FUNCTION_BLOCK "GCS7_E_MZMN"	// FB 22
TITLE = MZAG/MZAH Flowbalancer
//  
//COPYRIGHT:    (C) 1997 BY  BUHLER AG, CH-9240 UZWIL  SWITZERLAND
//
//PRODUCT:      GCS7
//
//TITLE:        Element MZMN (Profibus) 
//
//-------------------------------------------------------------------------
//
//IDENT:        AUTHOR:             DEPT:                      DATE:
//
//FB22.5.2      A. Egli             BASE                       09-Apr-2008
//              Disable Alarm 18 Battery Low
//FB22.5.1      A.Egli              CT3                        01-Dec-2005
//              Parameter Upload Change DBD86-->DBD88
//FB22.5.0      A.Egli              CT3                        05-Jan-2005
//              Parameter Upload (uses DB10)
//FB22.4.2      A.Egli              CT3                        17-Nov-2003
//              - Alarm 90: Fault not RemoteControl
//              - Send RecipeNr=0 as long StStopped or StFault
//FB22.4.1      A.Egli              CT3                        03-Nov-2003
//              - in local mode Change to StStopped, when OutComFault
//FB22.4.0      A. Egli             CT3                        17-Jun-2002
//              MZMN Micro Dosing
//              LC Alarm 14 (DPFault) =Log Text number 12
//FB22.1A       A. Egli             CT3                        16-Apr-1998
//              1st Release in S7
//
//-------------------------------------------------------------------------
//
//PURPOSE:      MANUAL : see [MZGxxMAN]
//
//RESTRICTIONS: S7
//              ACCU2: Pointer to dynamic datas of the element
//              ACCU1: Pointer to parameter datas of the element
//
//=======================================================
//Log Message: 
//------------------------------------------------------
//0     = Fault Cannceled
//1..79 = AlarmLC : Alarmnumber see manual of MEAF
//90    = Fault Remote Control
//91    = StStopped
//92    = StDosing
//93    = StEmptied
//94    = Timeout starting
//95    = Wrong value
//96    = Communication fault
//97    = 
//98    = 
//99    = Collected alarm
//
//=======================================================
//StCode:  State               
//------------------------------------------------------
//32    StFault                 
// 1    StStopped                   Stopped
//41    Stopped.HWStop              StStopped + InHWStop 
//51    Stopped.DPFault             StStopped + DPFault
// 2    StStarting              
// 3    StStarted               
// 7    StStopping              
//
AUTHOR : EA
FAMILY : GCS7LL
NAME : MZMN
VERSION : 5.1
VAR
  StCode : INT ;	//Element state code
  InEnable : BOOL ;	//Enable to run the element (manual and automatic mode)
  spare21 : BOOL ;
  spare22 : BOOL ;
  spare23 : BOOL ;
  CmdNewValue : BOOL ;	//Send new target values
  spare25 : BOOL ;
  spare26 : BOOL ;
  spare27 : BOOL ;
  CmdOff : BOOL ;	//Pulse to stop the element (manual mode)
  CmdOn : BOOL ;	//Pulse to start the element (manual mode)
  CmdNext : BOOL ;	//Pulse to start the element in automatic mode
  CmdFaultReset : BOOL ;	//Command to reset fault
  InLocal : BOOL ;	//1= Local mode (no fault by start with service switch)
  InManual : BOOL ;	//1= Manual / 0= Automatic
  InReport : BOOL ;	//Report of all state transitions
  spare0307 : BOOL ;
  InHWStop : BOOL ;	//HW stop is detected, no fault
  InDPFault : BOOL ;	//DP-Fault is detected, no fault
  InSimulation : BOOL ;	//Simulation with DPSim
  OutComFault : BOOL ;	//Communication fault
  spare44 : BOOL ;
  spare45 : BOOL ;
  spare46 : BOOL ;
  spare47 : BOOL ;
  StStopped : BOOL ;	//Element is stopped
  StStarting : BOOL ;	//Element is starting
  StStarted : BOOL ;	//Element is dosing
  StStopping : BOOL ;	//Element is stopping
  StFault : BOOL ;	//Element has a communication or device fault
  spare55 : BOOL ;
  spare56 : BOOL ;
  spare57 : BOOL ;
  InFlowrate : DINT ;	//Flowrate target value [0.1%]
  InRecipeNr : INT ;	//Is send to LC
  OutFlowrate : DINT ;	//Is read from LC [10g/h]
  OutRecipeNr : INT ;	//Is read from MEAF
  OutLCStep : INT ;	//Is read from MEAF
  OutAlarmNr : INT ;	//Is read from MEAF
  OutAlarmNrLog : INT ;	//Last textnumber send to log
  RecipeMZMN : STRUCT
   InRecipeNr : INT ;	//Recipe to read or write
   CmdSend : BOOL ;	//1= Send Dataset 136
   CmdRead : BOOL ;	//1= Read Dataset 136
   OutSendDone : BOOL ;	//Send is done
   OutReadDone : BOOL ;	//Read is done
   OutWrongValue : BOOL ;	//MEAF has recipe rejected
   Desity : INT ;	//de: Spezifisches Gewicht REC.DENS
   CorrectionFactor : INT ;	//de: Korrekturfactor REC.FACT
   NominalRate : INT ;	//de: Sollleistung REC.FLOS
   MixerFrequency : INT ;	//de: Frequenz Wirbler REC.MIX
   TypeRate : INT ;	//de: Volumetrische Typenleistung REC:FTYP
   AgitatorCutoutMode : INT ;	//de: Aussetzbetrieb Rührwerk REC.IOFF
   spare16 : INT ;
   spare18 : INT ;
  END_STRUCT ;
  Par : STRUCT
   ParObjectNo : INT ;	//Is used for communication with PC, e.g. for message
   ParMsgType : INT ;	//Is used for message (translation of state)
   ParHornCode : INT ;	//Is used by horn module
   ParLogOff : BOOL ;	//Report is off
   ParManual : BOOL ;	//Manual mode wihout interlocking
   ParFilter : STRUCT 	//Filter to alarm 1=Ignore alarm
    SumFault : BOOL ;	//de: Sammelalarm
    A05_24VToLow : BOOL ;
    A07ADRange : BOOL ;
    A08ADCalibration : BOOL ;
    A09ADFunction : BOOL ;
    A10ADSupply : BOOL ;
    A11AnalogInput : BOOL ;
    A12SerialInterface : BOOL ;
    A13RemoteControl : BOOL ;
    A16Printer : BOOL ;
    A25FrequenceConverter : BOOL ;
    A54Relais : BOOL ;
   END_STRUCT ;
   ParIOByteNr : INT ;	//PROFIBUS: Address of first input and output byte
   ParMonTime : INT ;	//Monitoring time starting and stopping
   OutMonTime : INT ;	//Monitoring time starting and stopping
   HelpFlags : STRUCT
    OutAlarmTimeOut : BOOL ;
    CmdNewValue : BOOL ;
    CmdFaultReset : BOOL ;
    OutFaultResetDone : BOOL ;
    OutTestNewAlarm : BOOL ;	//Aux. signal to retry fault message
    spare0007 : BOOL ;
    OutRelevantFault : BOOL ;
    OutNoAlarm : BOOL ;	//Alarmnumber 0 is read form LC
    OutFlagFaultResetDone : BOOL ;
    OutComFaultRead : BOOL ;
    OutComFaultSend : BOOL ;
   END_STRUCT ;
   Command : STRUCT
    Start : BOOL ;	//de: Start
    spare01 : BOOL ;
    spare02 : BOOL ;
    spare03 : BOOL ;
    spare04 : BOOL ;
    spare05 : BOOL ;
    spare06 : BOOL ;
    AcceptNewDataReady : BOOL ;	//de: Quittierung neue Werte Bereit
    spare10 : BOOL ;
    Recipe1 : BOOL ;	//MZMN: Command to select recipe 1
    Recipe2 : BOOL ;	//MZMN: Command to select recipe 2
    Recipe3 : BOOL ;	//MZMN: Command to select recipe 3
    Recipe4 : BOOL ;	//MZMN: Command to select recipe 4
    Recipe5 : BOOL ;	//MZMN: Command to select recipe 5
    Recipe6 : BOOL ;	//MZMN: Command to select recipe 6
    spare20 : BYTE ;
    CommandReady : BOOL ;	//de: Steuersignale gültig
    spare31 : BOOL ;
    spare32 : BOOL ;
    spare33 : BOOL ;
    spare34 : BOOL ;
    ResetAlarm : BOOL ;	//de: Alarm löschen
    NewSendData : BOOL ;	//de: Aenderung Sendedaten
    AcceptNewRcvData : BOOL ;	//de: Quittierung Aenderung Empfangsdatensatz
   END_STRUCT ;
   Status : STRUCT
    Operation : BOOL ;	//de: Betrieb
    spare01 : BOOL ;
    spare02 : BOOL ;
    spare03 : BOOL ;
    spare04 : BOOL ;
    spare05 : BOOL ;
    spare06 : BOOL ;
    NewDataReady : BOOL ;	//de: Neue Werte Bereit
    spare10 : BOOL ;
    Recipe1 : BOOL ;	//MZMN2 , Recipe 2 is active
    Recipe2 : BOOL ;	//MZMN3 , Recipe 3 is active
    Recipe3 : BOOL ;	//MZMN3 , Recipe 3 is active
    Recipe4 : BOOL ;	//MZMN4 , Recipe 4 is active
    Recipe5 : BOOL ;	//MZMN5 , Recipe 5 is active
    Recipe6 : BOOL ;	//MZMN6 , Recipe 6 is active
    spare20 : BYTE ;
    spare30 : BOOL ;
    spare31 : BOOL ;
    spare32 : BOOL ;
    RemoteControl : BOOL ;	//de: Sollwertvorgabe Remote
    WrongValue : BOOL ;	//de: Falscher Sollwert
    SumFault : BOOL ;	//de: Sammelalarm
    AcceptNewSendData : BOOL ;	//de: Quittierung Aenderung Sendedaten
    NewRcvData : BOOL ;	//de: Aenderung Empfangsdaten
   END_STRUCT ;
  END_STRUCT ;
END_VAR
VAR_TEMP
  tmpLOGvalue : WORD ;	//LOG value
  tmpCommand : INT ;
  tmpFault : BOOL ;
  tmpOff : BOOL ;
  tmpOn : BOOL ;
  tmpLocal : BOOL ;
  tmpLocalFault : BOOL ;
  tmpReport : BOOL ;
  tmpFlag : BOOL ;
  tmpLenDyn : DINT ;
  tmpAddrOutComFlags : DWORD ;	//Pointer to OutComFlags
  tmpWt : DINT ;
  tmpFilter : ARRAY  [0 .. 100 ] OF BOOL ;
  tmpAddrOffset : DINT ;
  tmpAddr : WORD ;
  tmpReturn : INT ;
  DPData : STRUCT
   StatusCommand : DWORD ;
   NrSndDataSet : BYTE ;	//de: Nummer Sendedatensatz
   IdxSndDataSet : BYTE ;	//de: Index Sendedatensatz
   NrRcvDataSet : BYTE ;	//de: Nummer Empfangsdatensatz
   IdxRcvDataSet : BYTE ;	//de: Index Empfangsdatensatz
   Data : ARRAY  [1 .. 4 ] OF DINT ;
  END_STRUCT ;
  Set001 : STRUCT
   FlowrateAc : DINT ;	//de: Istleistung kg/h
   spare4 : DINT ;	//de: Isttotalgewicht kg
   spare8 : DINT ;	//de: nochtlöschbarese Totalgewicht
   spare12 : BYTE ;
   RecipeNr : BYTE ;
   Step : BYTE ;
   AlarmNr : BYTE ;
  END_STRUCT ;
  tmpHornOn : BOOL ;
END_VAR
BEGIN
NETWORK
TITLE =  Start Global
      L     70;
      T     #tmpLenDyn;	//--> Len dynamic data in byte
      SET;
      R     #tmpHornOn;
NETWORK
TITLE = Filter
      LAR1  P##tmpFilter;
      L     0;
      T     D [AR1,P#0.0];	//tmpFilter[00..31]
      T     D [AR1,P#0.0];	//tmpFilter[32..63]
      T     D [AR1,P#0.0];	//tmpFilter[64..95]
      SET;	//[4.1]
      =     #tmpFilter[0];
      A     #Par.ParFilter.A05_24VToLow;
      =     #tmpFilter[5];
      A     #Par.ParFilter.A07ADRange;
      =     #tmpFilter[7];
      A     #Par.ParFilter.A08ADCalibration;
      =     #tmpFilter[8];
      A     #Par.ParFilter.A09ADFunction;
      =     #tmpFilter[9];
      A     #Par.ParFilter.A10ADSupply;
      =     #tmpFilter[10];
      A     #Par.ParFilter.A11AnalogInput;
      =     #tmpFilter[11];
      A     #Par.ParFilter.A12SerialInterface;
      =     #tmpFilter[12];
      =     #tmpFilter[14];	//[4.0]
      A     #Par.ParFilter.A13RemoteControl;
      =     #tmpFilter[13];
      A     #Par.ParFilter.A16Printer;
      =     #tmpFilter[16];
      SET;
      =     #tmpFilter[18];	//[5.2] Battery Low
      A     #Par.ParFilter.A25FrequenceConverter;
      =     #tmpFilter[25];
      A     #Par.ParFilter.A54Relais;
      =     #tmpFilter[54];
NETWORK
TITLE = PC Control
//=== Test Object number =====================
      L     "SYS_DirectCtrlDB".PC.ObjectNo;	//PCControl.ObjectNo
      L     #Par.ParObjectNo;	//Input ObjectNo
      <>I;
      JC    Ctrl;
//=== Test OType      ========================
      L     1022;	//Input object type
      L     "SYS_DirectCtrlDB".PC.ObjectType;	//PCControl.ObjectType
      <>I;
      JC    Ctrl;
//=== Test Handshake =========================
      A     "SYS_DirectCtrlDB".PC.Hsk.FExamine;	//Handshake.FExamine
      JC    pExa;
      A     "SYS_DirectCtrlDB".PC.Hsk.FDefineCmd;	//Handshake.FDefineCmd
      JC    pCmd;
      A     "SYS_DirectCtrlDB".PC.Hsk.FDefinePara;	//Handshake.FDefinePara
      JC    pPar;
pIni: L     2;	//FcInit
      UC    "SYS_DirectCtrl";
      JU    Ctrl;
// Write parameter 
pPar: LAR1  P#DBX 58.0;
      L     P##Par;
      L     DW#16#FFFFF;
      AD;
      +AR1;
      L     DBD [AR1,P#12.0];
      T     #Par.ParMonTime;
//Write new commands from PC to Interface of group 
pCmd: A     "SYS_DirectCtrlDB".PC.Cmd1[4];	//Cmd1[4]  =CmdNewValue
      S     #CmdNewValue;
      A     "SYS_DirectCtrlDB".PC.Cmd1[8];	//Cmd1[8]  =CmdOff
      S     #CmdOff;
      A     "SYS_DirectCtrlDB".PC.Cmd1[9];	//Cmd1[9]  =CmdOn
      S     #CmdOn;
      A     "SYS_DirectCtrlDB".PC.Cmd1[10];	//Cmd1[10] =CmdNext
      S     #CmdNext;
      A     "SYS_DirectCtrlDB".PC.Cmd1[11];	//Cmd1[11] =CmdFaultReset
      S     #CmdFaultReset;
      A     "SYS_DirectCtrlDB".PC.Cmd1[13];	//Cmd1[13] =CmdManualOn
      S     #InManual;
      A     "SYS_DirectCtrlDB".PC.Cmd2[13];	//Cmd2[13] =CmdManualOff
      R     #InManual;
      A     "SYS_DirectCtrlDB".PC.Cmd1[14];	//Cmd1[14] =CmdReportOn
      S     #InReport;
      A     "SYS_DirectCtrlDB".PC.Cmd2[14];	//Cmd2[14] =CmdReportOff
      R     #InReport;
//Define Value
      AN    "SYS_DirectCtrlDB".PC.Hsk.FDefineValue;	// PC.Hsk.FDefineValue
      ON    #InManual;
      JC    pIni;
      LAR1  P#DBX 58.0;
      L     DBD [AR1,P#6.0];
      T     #InFlowrate;
      L     DBW [AR1,P#10.0];
      T     #InRecipeNr;
      JU    pIni;
pExa: TAR2;	//Address dynamic datas
      T     "SYS_DirectCtrlDB".GC.InDynAddr;	//-->PCControl.GC.InDynAddr
      L     #tmpLenDyn;	//Length dynamic datas
      T     "SYS_DirectCtrlDB".GC.InDynLen;	//-->PCControl.GC.InDynLen
      L     0;
      T     "SYS_DirectCtrlDB".GC.InParaAddr;	//-->PCControl.GC.InParaAddr
      T     "SYS_DirectCtrlDB".GC.InParaLen;	//-->PCControl.GC.InParaLen
      L     1;	//Code FcExamine
      UC    "SYS_DirectCtrl";
      L     10;	//Revision
      T     "SYS_DirectCtrlDB".GC.Revision;
Ctrl: NOP   0;
NETWORK
TITLE = (Profibus) Read data and store Data 
      L     #Par.ParIOByteNr;
      T     #tmpAddr;
      A     #InSimulation;
      JC    rSim;
      CALL  "SIEMENS_DPRD_DAT" (
           LADDR                    := #tmpAddr,
           RET_VAL                  := #tmpReturn,
           RECORD                   := #DPData);
      L     #tmpReturn;
      L     0;
      <>I;
      =     #Par.HelpFlags.OutComFaultRead;
      JC    rcv0;
      JU    rDP;
//read from Simulation
rSim: R     #Par.HelpFlags.OutComFaultRead;
      A     "GCS7_Gr_SimDPtoImage";
      L     P#I 0.0;
      JC    rDB1;
      OPN   "TEST_IOSimuliInput";
      L     P#DBX 0.0;
rDB1: L     #Par.ParIOByteNr;
      SLD   3;
      +D;
      LAR1;
      L     D [AR1,P#0.0];
      T     #DPData.StatusCommand;
      L     B [AR1,P#4.0];
      T     #DPData.NrSndDataSet;
      L     B [AR1,P#5.0];
      T     #DPData.IdxSndDataSet;
      L     B [AR1,P#6.0];
      T     #DPData.NrRcvDataSet;
      L     B [AR1,P#7.0];
      T     #DPData.IdxRcvDataSet;
      L     D [AR1,P#8.0];
      T     #DPData.Data[1];
      L     D [AR1,P#12.0];
      T     #DPData.Data[2];
      L     D [AR1,P#16.0];
      T     #DPData.Data[3];
      L     D [AR1,P#20.0];
      T     #DPData.Data[4];
//==Copy Status===============
rDP:  L     #DPData.NrRcvDataSet;
      L     0;
      ==I;
      JC    R001;
      CALL  "SIEMENS_BLKMOV" (
           SRCBLK                   := #DPData.StatusCommand,
           RET_VAL                  := #tmpReturn,
           DSTBLK                   := #Par.Status);
      AN    #Par.Status.NewRcvData;
      A     #InSimulation;
      JC    rcv0;
//===============================
//Answer Dataset 001
      L     #DPData.NrRcvDataSet;
      L     1;
      <>I;
      JC    r11;	//[5.0]
      CALL  "SIEMENS_BLKMOV" (
           SRCBLK                   := #DPData.Data,
           RET_VAL                  := #tmpReturn,
           DSTBLK                   := #Set001);
      L     #Set001.FlowrateAc;
      T     #OutFlowrate;
      L     #Set001.RecipeNr;
      T     #OutRecipeNr;
      L     #Set001.Step;
      T     #OutLCStep;
//Reset old alarm flags with CmdFaultReset
      A     #Par.HelpFlags.OutFlagFaultResetDone;
      A     "SYS_Pulse1000ms";
      R     #Par.HelpFlags.OutFlagFaultResetDone;
      R     #Par.HelpFlags.OutFaultResetDone;
      S     #Par.HelpFlags.OutTestNewAlarm;
      L     0;
      L     #Set001.AlarmNr;
      ==I;
      =     #Par.HelpFlags.OutNoAlarm;
      <>I;
      O     #Par.ParFilter.SumFault;
      =     #tmpFilter[0];
//  keep old alalrm number
      A     #Par.HelpFlags.OutNoAlarm;
      A     #Par.HelpFlags.OutRelevantFault;
      AN    #Par.HelpFlags.OutTestNewAlarm;
      AN    #InLocal;
      AN    #InManual;
      JC    rA1;
      T     #OutAlarmNr;
rA1:  JU    R11;	//[5.0]
//===============================
//[5.0]--> LC Parameter 
//Reading dataset 11
R11:  L     "SYS_DirectCtrlLCDB".PC.ObjectNo;
      L     #Par.ParObjectNo;
      <>I;
      JC    R127;
      AN    "SYS_DirectCtrlLCDB".PC.Hsk.FExamineFirst;
      AN    "SYS_DirectCtrlLCDB".PC.Hsk.FExamineNext;
      JC    R127;
// -- Start Reading with Dataset 11
      L     11;
      T     #DPData.NrRcvDataSet;
      L     253;	//First
      A     "SYS_DirectCtrlLCDB".PC.Hsk.FExamineFirst;
      JC    rLC9;
      L     254;	//Next
rLC9: T     #DPData.IdxRcvDataSet;
      JU    rcv0;
//---Answer  dataset 11 ---
//---Answer  dataset 12 ---
r11:  L     #DPData.NrRcvDataSet;
      L     11;
      <>I;
      JC    rLCB;
// Answer Dataset 11
      L     '  ';
      T     "SYS_DirectCtrlLCDB".PC.Value[1];
      L     #DPData.Data[1];
      T     DB10.DBD 60;
      L     #DPData.Data[2];
      T     DB10.DBD 64;
      L     #DPData.Data[3];
      T     DB10.DBD 68;
      L     #DPData.Data[4];
      T     DB10.DBD 72;
      L     #DPData.IdxRcvDataSet;
      L     255;
      ==I;
      JC    rLCE;
      S     "SYS_DirectCtrlLCDB".GC.Set11Done;
      L     12;
      T     #DPData.NrRcvDataSet;
      L     0;
      T     #DPData.IdxRcvDataSet;
      JU    rcv0;	//--> Read dataset 12
// Answer Dataset 12
rLCB: L     #DPData.NrRcvDataSet;
      L     12;
      <>I;
      JC    r127;
      L     #DPData.Data[1];
      T     DB10.DBD 76;
      L     #DPData.Data[2];
      T     DB10.DBD 80;
      L     #DPData.Data[3];
      T     DB10.DBD 84;
      L     #DPData.Data[4];
      T     DB10.DBD 88;
      AN    "SYS_DirectCtrlLCDB".GC.Set11Done;
      JC    R127;
rLCE: L     12;
      CALL  "SYS_DirectCtrl";
      JU    R127;
//<--[5.0]
//===============================
//Answer  dataset 127
r127: L     #DPData.NrRcvDataSet;
      L     127;
      <>I;
      JC    r128;
      JU    R128;
//===============================
//Answer  dataset 128
r128: JU    r136;
//===============================
//Answer  dataset 136
r136: L     #DPData.NrRcvDataSet;
      L     136;
      <>I;
      JC    R001;	// =no valide answer read dataset 001
      L     #RecipeMZMN.InRecipeNr;
      L     #DPData.IdxRcvDataSet;
      ==I;
      JCN   R001;
      R     #RecipeMZMN.CmdRead;
      S     #RecipeMZMN.OutReadDone;
      L     #DPData.Data[1];
      T     #RecipeMZMN.CorrectionFactor;
      SRD   16;
      T     #RecipeMZMN.Desity;
      L     #DPData.Data[2];
      T     #RecipeMZMN.NominalRate;
      L     #DPData.Data[3];
      T     #RecipeMZMN.TypeRate;
      SRD   16;
      T     #RecipeMZMN.MixerFrequency;
      L     #DPData.Data[4];
      L     W#16#FFFF;
      AW;
      SRD   8;
      T     #RecipeMZMN.AgitatorCutoutMode;
      JU    R001;
//===============================
//Read Dataset 001
R001: L     1;
      T     #DPData.NrRcvDataSet;
      L     0;
      T     #DPData.IdxRcvDataSet;
      A     #Par.HelpFlags.OutFaultResetDone;
      AN    "SYS_Pulse1000ms";
      S     #Par.HelpFlags.OutFlagFaultResetDone;
      JU    rcv0;
//===============================
//Read Dataset 127
R127: L     127;
      T     #DPData.NrRcvDataSet;
      L     0;
      T     #DPData.IdxRcvDataSet;
      JU    rcv0;
//===============================
//Read Dataset 128
R128: JU    R136;
//===============================
//Read Dataset 136
R136: AN    #RecipeMZMN.CmdRead;
      JC    R001;
      L     136;
      T     #DPData.NrRcvDataSet;
      L     #RecipeMZMN.InRecipeNr;
      T     #DPData.IdxRcvDataSet;
      JU    rcv0;
//===============================
rcv0: NOP   0;
      NOP   0;
NETWORK
TITLE = (Profibus) Status to ASW
      A     #Par.HelpFlags.OutComFaultRead;
      O     #Par.HelpFlags.OutComFaultSend;
      =     #OutComFault;
//=======================================
//Init in local mode  
//=======================================
      AN    #InLocal;
      AN    #InManual;
      ON    #OutComFault;
      JC    alJL;
      L     0;
      T     #OutFlowrate;
alJL: NOP   0;
      NOP   0;
NETWORK
TITLE =  All State Init
//===Clear tmp Variable
//===Global Group Orders===
      A     "GCS7_Gr_OutManualOn";	//Global.OutManualOn
      S     #InManual;
      A     "GCS7_Gr_OutManualOff";	//Global.OutManualOff
      R     #InManual;
      A     #InManual;
      S     "GCS7_Gr_InManual";	//Global.InManualMode
//---Report is on---
      O     "GCS7_Gr_OutReportAll";	//---Global OutReportAll
      O     #InReport;
      =     #tmpReport;
//---FaultReset is on---
      A     "GCS7_Gr_OutFaultReset";	//Gr.OutFaultReset
      S     #CmdFaultReset;
//---Local---
      A     #InLocal;
      AN    #InManual;
      =     #tmpLocalFault;
      A     #tmpLocalFault;
      O     #InHWStop;
      O     #InDPFault;
      =     #tmpLocal;
//---Off---
      AN    #InManual;
      ON    #Par.ParManual;
      AN    #InEnable;
      O     #tmpLocal;
      O     #CmdOff;
      =     #tmpOff;
//---On---
      A     #CmdNext;
      AN    #InManual;
      O     #CmdOn;
      AN    #tmpOff;
      =     #tmpOn;
//--- Send Recipe
      A     #RecipeMZMN.CmdSend;
      R     #RecipeMZMN.OutSendDone;
//--- Read Recipe
      A     #RecipeMZMN.CmdRead;
      R     #RecipeMZMN.OutReadDone;
//--- tmpFault   
// Time out
      AN    #StStarting;
      AN    #StStopping;
      AN    #StFault;
      R     #Par.HelpFlags.OutAlarmTimeOut;
      JC    inJ1;
      A     #Par.HelpFlags.OutAlarmTimeOut;
      O     #StFault;
      JC    inJ1;
      L     0;
      L     #Par.OutMonTime;
      >I;
      =     #Par.HelpFlags.OutAlarmTimeOut;
      AN    "GCS7_Gr_OutTick200ms";	// Global Tick 200ms
      JC    inJ1;
      +     -2;	// Decrement all 200ms
      T     #Par.OutMonTime;
inJ1: NOP   0;
//=======================================
//Fault   
//=======================================
      LAR1  P##tmpFilter;
      L     #OutAlarmNr;
      +AR1;	//Pointer to #tmpFilter[OutAlarmNumber]
      L     #OutAlarmNr;
      L     0;
      <>I;
      AN    L [AR1,P#0.0];	//#tmpFilter[OutAlarmNumber]
      =     #Par.HelpFlags.OutRelevantFault;
      A     #Par.HelpFlags.OutRelevantFault;
      O     #OutComFault;
      O     #Par.HelpFlags.OutAlarmTimeOut;
      O     #Par.Status.WrongValue;
      ON    #Par.Status.RemoteControl;	//[4.2]
      AN    #tmpLocal;
      =     #tmpFault;
      NOP   0;
NETWORK
TITLE = (Profibus) Prepare Command for MEAF
//==============================
      A     #Par.Status.AcceptNewSendData;
      A     #Par.Command.ResetAlarm;
      R     #Par.Command.ResetAlarm;
      S     #Par.HelpFlags.OutFaultResetDone;
      A     #CmdFaultReset;
      AN    #Par.Status.AcceptNewSendData;
      R     #CmdFaultReset;
      S     #Par.Command.ResetAlarm;
      R     #Par.HelpFlags.OutAlarmTimeOut;
//================================
      A     #tmpOn;
      AN    #Par.HelpFlags.CmdNewValue;
      S     #Par.Command.Start;
      A     #StFault;
      A     #Par.HelpFlags.OutNoAlarm;
      O     #tmpOff;
      R     #Par.Command.Start;
//==============================
      A     #Par.Status.NewDataReady;
      =     #Par.Command.AcceptNewDataReady;
//==============================
      SET;
      =     #Par.Command.CommandReady;
//==============================
      A     #Par.Status.NewRcvData;
      =     #Par.Command.AcceptNewRcvData;
//==============================
      AN    #Par.Status.AcceptNewSendData;
      =     #Par.Command.NewSendData;
//==============================
//Command MZMN 
      L     #InRecipeNr;
      L     1;
      ==I;
      =     #Par.Command.Recipe1;
      L     #InRecipeNr;
      L     2;
      ==I;
      =     #Par.Command.Recipe2;
      L     #InRecipeNr;
      L     3;
      ==I;
      =     #Par.Command.Recipe3;
      L     #InRecipeNr;
      L     4;
      ==I;
      =     #Par.Command.Recipe4;
      L     #InRecipeNr;
      L     5;
      ==I;
      =     #Par.Command.Recipe5;
      L     #InRecipeNr;
      L     6;
      ==I;
      =     #Par.Command.Recipe6;
      NOP   0;
NETWORK
TITLE = (Profibus) Send Data
//======================================================
//Test Send Dataset 000 done
      L     #DPData.NrSndDataSet;
      L     0;
      <>I;
      JC    s128;
      JU    S128;	//-->send 128
//------------------------------------------------
//Test Send Dataset 128 done
s128: L     #DPData.NrSndDataSet;
      L     128;
      <>I;
      JC    s136;
      AN    #Par.Status.WrongValue;
      A     #Par.HelpFlags.CmdNewValue;
      A     #CmdNewValue;
      R     #Par.HelpFlags.CmdNewValue;
      R     #CmdNewValue;
      JU    S136;	//-->Send 136
//------------------------------------------------
//Test Send Dataset 136 done
s136: L     #DPData.NrSndDataSet;
      L     136;
      <>I;
      JC    S000;
      L     #DPData.IdxSndDataSet;
      L     #RecipeMZMN.InRecipeNr;
      ==I;
      JCN   S128;	//-->Send 128
      A     #Par.Status.WrongValue;
      S     #RecipeMZMN.OutWrongValue;
      AN    #Par.Status.WrongValue;
      R     #RecipeMZMN.CmdSend;
      S     #RecipeMZMN.OutSendDone;
      R     #RecipeMZMN.OutWrongValue;
      JU    S128;	//-->Send 128
//==================================================
//Send Dataset 128
S128: A     #CmdNewValue;
      =     #Par.HelpFlags.CmdNewValue;
      L     128;
      T     #DPData.NrSndDataSet;
      L     0;
      T     #DPData.IdxSndDataSet;
      L     #InFlowrate;
      SLD   16;
      T     #DPData.Data[1];
      L     0;
      T     #DPData.Data[2];
      L     0;
      T     #DPData.Data[3];
      A     #StStopped;	//[4.2]
      O     #StFault;	//[4.2]
      L     0;	//[4.2]
      JC    snJ8;	//[4.2]
      L     #InRecipeNr;
      SLD   16;
snJ8: T     #DPData.Data[4];	//-->Byte 21
      JU    send;
//======================================================
//Send Dataset 136
S136: AN    #RecipeMZMN.CmdSend;
      JC    S000;
      L     136;
      T     #DPData.NrSndDataSet;
      L     #RecipeMZMN.InRecipeNr;
      T     #DPData.IdxSndDataSet;
      L     #RecipeMZMN.Desity;
      SLD   16;
      L     #RecipeMZMN.CorrectionFactor;
      OD;
      T     #DPData.Data[1];
      L     #RecipeMZMN.NominalRate;
      T     #DPData.Data[2];
      L     #RecipeMZMN.MixerFrequency;
      SLD   16;
      L     #RecipeMZMN.TypeRate;
      OD;
      T     #DPData.Data[3];
      L     #RecipeMZMN.AgitatorCutoutMode;
      SLD   8;
      T     #DPData.Data[4];
      JU    send;
//======================================================
//Send Dataset 0
S000: L     0;
      T     #DPData.NrSndDataSet;
      L     0;
      T     #DPData.IdxSndDataSet;
send: CALL  "SIEMENS_BLKMOV" (
           SRCBLK                   := #Par.Command,
           RET_VAL                  := #tmpReturn,
           DSTBLK                   := #DPData.StatusCommand);
      A     #InSimulation;
      JC    sSim;
      CALL  "SIEMENS_DPWR_DAT" (
           LADDR                    := #tmpAddr,
           RECORD                   := #DPData,
           RET_VAL                  := #tmpReturn);
      L     #tmpReturn;
      L     0;
      <>I;
      =     #Par.HelpFlags.OutComFaultSend;
      JU    DP_C;
//write to Simulation
sSim: R     #Par.HelpFlags.OutComFaultSend;
      A     "GCS7_Gr_SimDPtoImage";
      L     P#Q 0.0;
      JC    rDB2;
      OPN   "TEST_IOSimuliOutput";
      L     P#DBX 0.0;
rDB2: L     #Par.ParIOByteNr;
      SLD   3;
      +D;
      LAR1;
      L     #DPData.StatusCommand;
      T     D [AR1,P#0.0];
      L     #DPData.NrSndDataSet;
      T     B [AR1,P#4.0];
      L     #DPData.IdxSndDataSet;
      T     B [AR1,P#5.0];
      L     #DPData.NrRcvDataSet;
      T     B [AR1,P#6.0];
      L     #DPData.IdxRcvDataSet;
      T     B [AR1,P#7.0];
      L     #DPData.Data[1];
      T     D [AR1,P#8.0];
      L     #DPData.Data[2];
      T     D [AR1,P#12.0];
      L     #DPData.Data[3];
      T     D [AR1,P#16.0];
      L     #DPData.Data[4];
      T     D [AR1,P#20.0];
DP_C: NOP   0;
NETWORK
TITLE = States
//===State machine===
      A     #StStopped;
      JC    S0;
      A     #StStarting;
      JC    S1;
      A     #StStarted;
      JC    S2;
      A     #StStopping;
      JC    S3;
      A     #StFault;
      JC    S4;
      S     #StStopped;	//Init
      JU    S0;
NETWORK
TITLE =  StStopped
xxS0: S     #StStopped;
      R     #StStarted;
      JU    LOGX;
S0:   A     #tmpFault;
      S     #tmpHornOn;
      R     #StStopped;
      JC    xxS4;	////--> Transition to StFault
      A     #tmpOn;
      O     #Par.Status.Operation;
      AN    #OutComFault;	//[4.1]
      R     #StStopped;
      JC    xxS1;	//--> Transition to StStarting
      JU    OUT;
NETWORK
TITLE =  StStarting
xxS1: S     #StStarting;
      R     #Par.HelpFlags.OutAlarmTimeOut;
      L     #Par.ParMonTime;
      T     #Par.OutMonTime;
      JU    OUT;
S1:   A     #tmpFault;	//Condition for StFault
      R     #StStarting;
      JC    xxS4;	//--> Transition to StFault
      A     #tmpOff;
      R     #StStarting;
      JC    xxS3;	//--> Transition to StStopping
      A     #Par.Status.Operation;
      R     #StStarting;
      JC    xxS2;	//--> Transition to StStarted
      JU    OUT;
NETWORK
TITLE =  StStarted
xxS2: S     #StStarted;
      R     #StStopped;
      JU    LOGX;
S2:   A     #tmpFault;	//Condition for StFault/StFalse
      S     #tmpHornOn;
      R     #StStarted;
      JC    xxS4;	//--> Transition to StFault
      A     #tmpOff;
      ON    #Par.Status.Operation;
      O     #OutComFault;	//[4.1]
      R     #StStarted;
      JC    xxS3;	//--> Transition to StStopping
      JU    OUT;
NETWORK
TITLE =  StStopping
xxS3: S     #StStopping;
      R     #Par.HelpFlags.OutAlarmTimeOut;
      L     #Par.ParMonTime;
      T     #Par.OutMonTime;
      A     #StFault;
      R     #StFault;
      JC    LOGC;	//-->Message Operator ('fault cancelled' )
//-----------------------------------
//--> Transition to StFault
S3:   A     #tmpFault;
      AN    #tmpLocal;
      S     #tmpHornOn;
      R     #StStopping;
      JC    xxS4;	//-->Transition to StFault
//-----------------------------------
//--> Transition to StStarting
      A     #tmpOn;
      R     #StStopping;
      JC    xxS1;	//-->Transition to StStarting 
//-----------------------------------
//--> Transition to StStopped
      AN    #tmpFault;	//Transition to StFaulte
      AN    #Par.Status.Operation;
      O     #OutComFault;	//[4.1]
      R     #StStopping;
      JC    xxS0;	//-->Transition to StStopped 
      JU    OUT;
NETWORK
TITLE =  FAULT
// State Fault
S4:   AN    #tmpFault;	//---Condition for StStopping
      A     #Par.HelpFlags.OutTestNewAlarm;
      O     #tmpLocalFault;
      JC    xxS3;	// Transition to StStopping
      A     #Par.HelpFlags.OutTestNewAlarm;
      JC    xxS4;
      JU    OUT;
NETWORK
TITLE = LOG
xxS4: S     #tmpHornOn;
      S     #StFault;
      R     #Par.HelpFlags.OutFaultResetDone;
      R     #Par.HelpFlags.OutTestNewAlarm;
      L     #Par.ParMonTime;
      T     #Par.OutMonTime;
//Alarm Communication
      L     B#(1, 96);
      A     #OutComFault;
      JC    LOG;
//Tiemout
      A     #Par.HelpFlags.OutAlarmTimeOut;
      L     B#(1, 94);	// Message ('fault timeout')
      JC    LOG;
//Alarm-Nr 1..80
      L     0;
      L     #OutAlarmNr;
      ==I;
      JC    LOG2;
      L     B#(1, 0);
      OW;
      JU    LOG;	//Alarms 1..80
//Fault Wrong Value
LOG2: L     B#(1, 90);	// Message ('fault DP Mode')   //[4.2]
      AN    #Par.Status.RemoteControl;	//[4.2]
      JC    LOG;	//[4.2]
//Fault Wrong Value
      A     #Par.Status.WrongValue;
      L     B#(1, 95);	// Message ('fault wrong value')
      JC    LOG;
//Collected Alarm
      L     B#(1, 99);	// Message ('fault collected alarm')
      JU    LOG;
//===============================================
//State Transition
LOGX: AN    #tmpReport;
      JC    OUT;
      A     #StStopped;
      L     B#(4, 91);	//Message ('Stopped')
      JC    LOG;
      A     #StStarted;
      L     B#(4, 92);	//Message ('Dosing')
      JC    LOG;
      JU    OUT;
LOGC: L     B#(4, 0);	//Message ('fault cancelled')
LOG:  A     #Par.ParLogOff;	//---Set LOG Message
      JC    SAVE;
      T     #tmpLOGvalue;
      L     W#16#FF;
      AW;
      T     #OutAlarmNrLog;
      CALL  "GCS7_LogConvert" (
           ObjectNo                 := #Par.ParObjectNo,
           MsgType                  := #Par.ParMsgType,
           ClassMsgTxt              := #tmpLOGvalue,
           OType                    := 1026);	//LOG Message Converter / Entry / Contains Class and TextNo
SAVE: NOP   0;
OUT:  NOP   0;
NETWORK
TITLE = Global End
      SET;	//---Clear all commands
      R     #CmdOff;
      R     #CmdOn;
      R     #CmdNext;
//---Horn On-----------------------------
      AN    #tmpHornOn;
      JC    glJ1;
      S     "GCS7_Gr_InFaultFlag";	// Gr.InFaultFlag
      CALL  "SYS_Horn_Code" (
           FcCode                   := 1,
           ParObjectType            := 1022,
           ParObjectNo              := #Par.ParObjectNo,
           ParHornCode              := #Par.ParHornCode);
glJ1: NOP   0;
//--Output for group 
      AN    #InLocal;
      O     #InManual;
      A     #InDPFault;
      S     "GCS7_Gr_InDPFault";
      AN    #InLocal;
      O     #InManual;
      A     #InHWStop;
      S     "GCS7_Gr_InHWStop";
NETWORK
TITLE = State Code
//--Stopped, Substate ---
      AN    #StStopped;
      JC    STC2;
      L     41;	//Code: StStopped.HWStop
      A     #InHWStop;
      JC    STC;
      L     51;	//Code: StStopped.DPFault
      A     #InDPFault;
      JC    STC;
      L     1;	// Code: stopped
      JC    STC;
//--------------------
STC2: L     2;	//Code: StStarting
      A     #StStarting;
      JC    STC;
      L     3;	//Code: StStarted
      A     #StStarted;
      JC    STC;
      L     7;	//Code: StStopping
      A     #StStopping;
      JC    STC;
      L     32;	//Code: fault
STC:  L     #StCode;	//Old state code
      TAK;
      T     #StCode;	//Save state code
      <>I;
      L     3;	//Load code for CBit methode
      CC    "SYS_CBitCtrl";
NETWORK
TITLE =  Store LC data
      BEU;
END_FUNCTION_BLOCK

FUNCTION_BLOCK "GCS7_E_MYEB"	// FB 23
TITLE = MYEB
//  
//COPYRIGHT:    (C) 1997  BUHLER AG, CH-9240 UZWIL, SWITZERLAND
//
//PRODUCT:      GCS7
//
//TITLE:        Element MYEB Moisture Control Unit
//
//-------------------------------------------------------------------------
//
//IDENT:        AUTHOR:             DEPT:                      DATE:
//
//FB23.5.0      A.Egli              CT3                        05-Jan-2005
//              Parameter Upload (uses DB10)
//FB23.4.1      A. Egli             CT3                        19-Nov-2004
//              With CmdNewJob immediately clear actual values 
//FB23.4.0      A. Egli             CT3                        17-Jun-2002
//              New Release with one block 
//FB23.2.2      A. Egli             CT3                        17-Mar-2000
//              Length for answer telegram
//FB23.2.1      S. Kalberer         CT3                        06-Dec-1999
//              No horn if InLocal
//FB23.2A       A. Egli             CT3                        04-Mai-1998
//              StFault = StCode 32
//FB23.1B       A.Egli              AEE61                      15-Apr-1998
//              RS485
//FB23.1A       S. Kalberer         AEE61                      17-Jul-1997
//              1st Release in S7
//
//-------------------------------------------------------------------------
//
//PURPOSE:      MANUAL : see [MYExxMAN]
//
//RESTRICTIONS: S7
//              ACCU2: Pointer to dynamic datas of the element
//              ACCU1: Pointer to parameter datas of the element
//
//-------------------------------------------------------------------------
//=======================================================
//Log Message: 
//------------------------------------------------------
//  1  software timer overflow     = #OutLCAlarm.SoftwareTimerOverflow
//  2  positive limit band exceeded= #OutLCAlarm.PosLimitBand
//  3  negative limit band exceeded= #OutLCAlarm.NegLimitBand
//  4  fault cancelled
//  5  MOZE function alarm         = #OutLCAlarm.MOZEFncAlarm
//  6  MOZE communication alarm    = #OutLCAlarm.MOZEComAlarm
//  7  MOZE configuration alarm    = #OutLCAlarm.MOZEConfigAlarm
//  8  MOZE minimum setpoint alarm = #OutLCAlarm.MOZEMinSetPointAlarm
//  9  MOZE maximum setpoint alarm = #OutLCAlarm.MOZEMaxSetPointAlarm
//  10 MYFB function alarm         = #OutLCAlarm.MYFBFncAlarm
//  11 MYFB communication alarm    = #OutLCAlarm.MYFBComAlarm
//  12 MYFB configuration alarm    = #OutLCAlarm.MYFBConfigAlarm
//  13 MYFB measurement alarm      = #OutLCAlarm.MYFBMeasureAlarm
//  14 fault MYEB communication    = OutComFault
//  15 flow meter function alarm   = #OutLCAlarm.FlowFncAlarm
//  16 flow meter communication alarm= #OutLCAlarm.FlowComAlarm
//  17 flow meter configuration alarm= #OutLCAlarm.FlowConfigAlarm
//
//=======================================================
//StCode:  State               
//------------------------------------------------------
//32    StFault           
// 3    StOk              
// 5    StFalse           
//45    StFalse.HWStop           StFalse + InHWStop
//55    StFalse.DPFault          StFalse + InDPFault
//
//
AUTHOR : EA
FAMILY : GCS7LL
NAME : MYEB
VERSION : 5.0
VAR
  StCode : INT ;	//Element state code
  spare0200 : BOOL ;
  InLimitOn : BOOL ;	//Signal to activate alarm limit band
  spare0202 : BOOL ;
  spare0203 : BOOL ;
  CmdNewValue : BOOL ;	//Send new target value to MYEB
  CmdNewJob : BOOL ;	//Clear actual values of MYEB
  InpProductAlarm : BOOL ;	//DI product alarm
  InpGroupAlarm : BOOL ;	//DI group alarm
  spare0300 : BOOL ;
  spare0301 : BOOL ;
  spare0302 : BOOL ;
  CmdFaultReset : BOOL ;	//Command to reset fault
  InLocal : BOOL ;	//1= Local mode (no fault by start with service switch)
  InManual : BOOL ;
  spare0306 : BOOL ;
  spare0307 : BOOL ;
  InHWStop : BOOL ;	//HW stop is detected, no fault
  InDPFault : BOOL ;	//DP-Fault is detected, no fault
  OutComFault : BOOL ;	//Communication fault
  OutFaultResetDone : BOOL ;	//Aux. signal fault reset done
  OutNewValueActive : BOOL ;	//Aux. signal new values active
  spare0405 : BOOL ;
  spare0406 : BOOL ;
  OutRequestActive : BOOL ;	//Aux. signal request active
  spare0500 : BOOL ;
  spare0501 : BOOL ;
  StOk : BOOL ;	//Element is ok
  spare0503 : BOOL ;
  StFault : BOOL ;	//Element has a communication or device fault
  StFalse : BOOL ;	//Element is in local mode and has a fault
  InStartValue : DINT ;	//Is send to LC
  InFlowrateProduct : DINT ;	//Is send to LC [kg/h]
  InTargetValue : DINT ;	//Is send to LC [0.1 l/h] or [0.01%]
  InLimitPos : INT ;	//Is send to LC [0.01%]
  InLimitNeg : INT ;	//Is send to LC [0.01%]
  InOffsetMoisture : DINT ;	//Is send to LC [0.01%]
  InDosingMax : DINT ;	//Is send to LC [0.1 l/h]
  InProductGroup : INT ;	//Is send to LC [0..99]
  OutTargetValue : DINT ;	//Is read from LC [0.01%]
  OutActualValue : DINT ;	//Is read from LC [0.01%]
  OutFlowrateProduct : DINT ;	//Is read from LC [kg/h]
  OutTotalProduct : DINT ;	//Is read from LC [kg]
  OutFlowrateWaterTarget : DINT ;	//Is read from LC [0.1 l/h]
  OutFlowrateWater : DINT ;	//Is read from LC [0.1 l/h]
  OutTotalWater : DINT ;	//Is read from LC [0.1 l]
  OutAlarmNr : INT ;	//Is read from LC
  OutNotErasableWater : DINT ;	//Is read from LC [0.1 l]
  spare6600 : DINT ;
  spare7000 : INT ;
  OutAlarmNrLog : INT ;	//Last textnumber send to log
  Par : STRUCT
   ParObjectNo : INT ;	//Is used for communication with PC, e.g. for message
   ParMsgType : INT ;	//Is used for message (translation of state)
   ParHornCode : INT ;	//Is used by horn module
   ParLogOff : BOOL ;	//Report is off
   ParFilter : STRUCT 	//Filter to alarm 1=Ignore alarm
    spare00 : BOOL ;
    SoftwareTimerOverflow : BOOL ;	//[A] Software timer overflow
    PosLimitBand : BOOL ;	//[P] Positive limit band exceeded
    NegLimitBand : BOOL ;	//[P] Negative limit band exceeded
    spare04 : BOOL ;
    MOZEFncAlarm : BOOL ;	//[A] MOZE function alarm
    MOZEComAlarm : BOOL ;	//[A] MOZE communication alarm
    MOZEConfigAlarm : BOOL ;	//[A] MOZE configuration alarm
    MOZEMinSetPointAlarm : BOOL ;	//[P] MOZE setpoint limiting minimum alarm
    MOZEMaxSetPointAlarm : BOOL ;	//[P] MOZE setpoint limiting maximum alarm
    MYFBFncAlarm : BOOL ;	//[A] MYFB function alarm
    MYFBComAlarm : BOOL ;	//[A] MYFB communication alarm
    MYFBConfigAlarm : BOOL ;	//[A] MYFB configuration alarm
    MYFBMeasureAlarm : BOOL ;	//[A] MYFB measurement alarm
    spare16 : BOOL ;
    FlowFncAlarm : BOOL ;	//[A] Flow meter function alarm
    FlowComAlarm : BOOL ;	//[A] Flow meter communication alarm
    FlowConfigAlarm : BOOL ;	//[A] Flow meter configuration alarm
   END_STRUCT ;
   ParComFlags : STRUCT
    spare00 : BYTE ;
    Without_O : BOOL ;	//Start value
    Without_Q : BOOL ;	//Product flowrate
    Without_T : BOOL ;	//Target value
    Without_U : BOOL ;	//Limits
    Without_F : BOOL ;	//Offset moisture
    Without_X : BOOL ;	//Dosing maximum
    Without_R : BOOL ;	//Product group
   END_STRUCT ;
   ParComDB : INT ;	//Communication DB
   ParLCIdx : INT ;	//Index of data record
   ParLCAddr : INT ;	//Address of LC
   OutLCState : STRUCT 	//Is read from LC
    spare00 : BYTE ;
    HostActive : BOOL ;	//Host control active
    DosingRelease : BOOL ;	//Dosing release
    AlarmActive : BOOL ;	//Alarm active
    RegulationOn : BOOL ;	//Regulation on
    PowerFailure : BOOL ;	//Power failure
    LoopActive : BOOL ;	//Loop active 1:RUN/ 0:SUSPEND
    LimitActive : BOOL ;	//Alarm limit band control active
    spare17 : BOOL ;
   END_STRUCT ;
   OutLCAlarm : STRUCT 	//Alarm bit mask of OutAlarmNumber
    spare00 : BOOL ;
    SoftwareTimerOverflow : BOOL ;	//[A] Software timer overflow
    PosLimitBand : BOOL ;	//[P] Positive limit band exceeded
    NegLimitBand : BOOL ;	//[P] Negative limit band exceeded
    spare04 : BOOL ;
    MOZEFncAlarm : BOOL ;	//[A] MOZE function alarm
    MOZEComAlarm : BOOL ;	//[A] MOZE communication alarm
    MOZEConfigAlarm : BOOL ;	//[A] MOZE configuration alarm
    MOZEMinSetPointAlarm : BOOL ;	//[P] MOZE setpoint limiting minimum alarm
    MOZEMaxSetPointAlarm : BOOL ;	//[P] MOZE setpoint limiting maximum alarm
    MYFBFncAlarm : BOOL ;	//[A] MYFB function alarm
    MYFBComAlarm : BOOL ;	//[A] MYFB communication alarm
    MYFBConfigAlarm : BOOL ;	//[A] MYFB configuration alarm
    MYFBMeasureAlarm : BOOL ;	//[A] MYFB measurement alarm
    spare16 : BOOL ;
    FlowFncAlarm : BOOL ;	//[A] Flow meter function alarm
    FlowComAlarm : BOOL ;	//[A] Flow meter communication alarm
    FlowConfigAlarm : BOOL ;	//[A] Flow meter configuration alarm
   END_STRUCT ;
   OutStateTarget : STRUCT 	//Command for LC, is send to LC
    spare00 : BYTE ;
    spare10 : BOOL ;
    spare11 : BOOL ;
    AlarmReset : BOOL ;	//Alarm reset
    spare13 : BOOL ;
    ClearPowerFlag : BOOL ;	//Clear powerfailure flag
    ClearLoopDatas : BOOL ;	//Clear loop datas
    LimitActive : BOOL ;	//Alarm limit band active
    spare17 : BOOL ;
   END_STRUCT ;
   OutComFlags : STRUCT 	//Flags for communication
    c_Done : BOOL ;	//Actual product data
    g_Done : BOOL ;	//Not erasable total of MOZE
    O_Done : BOOL ;	//Start value
    Q_Done : BOOL ;	//Product flowrate
    T_Done : BOOL ;	//Target value
    U_Done : BOOL ;	//Limits
    F_Done : BOOL ;	//Offset moisture
    X_Done : BOOL ;	//Dosing maximum
    R_Done : BOOL ;	//Product group
   END_STRUCT ;
  END_STRUCT ;
END_VAR
VAR_TEMP
  tmpLOGvalue : WORD ;	//LOG value
  tmpCommand : INT ;
  tmpFBNO : INT ;	//Number of the actual FB
  tmpFault : BOOL ;
  tmpComActive : BOOL ;	//Put or get is in queue
  tmpClearCmdFlag : BOOL ;	//Clear pattern Commands
  tmpLenDyn : DINT ;
  tmpAddrParFilter : DWORD ;	//Pointer to ParFilter
  tmpAddrOutLCState : DWORD ;	//Pointer to OutLCState
  tmpAddrOutLCAlarm : DWORD ;	//Pointer to OutLCAlarm
  tmpAddrOutStateTarget : DWORD ;	//Pointer to OutLCStateTarget
  tmpComDB : INT ;
  tmpLocal : BOOL ;
  tmpAddrOffset : DINT ;
END_VAR
BEGIN
NETWORK
TITLE =  Start Global
      L     23;
      T     #tmpFBNO;
      L     102;
      T     #tmpLenDyn;	//--> Len dynamic data in byte
      TAR2;
      L     DW#16#FFFFFF;
      AD;
      T     #tmpAddrOffset;
      L     P##Par;
      L     #tmpAddrOffset;
      +D;
      LAR1;
      L     P#8.0;	//Offset ParFilter
      +D;
      T     #tmpAddrParFilter;	//-->Pointer to ParFilter
      TAR1;
      L     P#20.0;	//P##Par.Par.OutLCState
      +D;
      T     #tmpAddrOutLCState;	//-->Pointer to OutLCState
      TAR1;
      L     P#22.0;	//P##Par.OutLCAlarm
      +D;
      T     #tmpAddrOutLCAlarm;	//-->Pointer to OutLCAlarm
      TAR1;
      L     P#26.0;	//P##Par.OutStateTarget
      +D;
      T     #tmpAddrOutStateTarget;	//-->Pointer to OutStateTarget
      L     #Par.ParComDB;
      T     #tmpComDB;
NETWORK
TITLE =  Call back function
//*****This functions are called by FBxxx (COM) ******
      OPN   DB [#tmpComDB];
      L     0;
      L     DBW 32;	//COM.Element.CODE;
      ==I;
      JC    PC;
      L     DBB 76;	//COM.Telegram.Command;
      T     #tmpCommand;
      L     1;
      L     DBW 32;	//COM.Element.CODE;
      ==I;
      JC    Send;
      L     2;
      ==I;
      JC    Rcv;
      L     4;	//NAK
      L     DBW 32;	//COM.Element.CODE;
      ==I;
      S     #OutComFault;	//fault MYEB communication
      JU    STOR;
//Read telegram length
Send: L     #tmpCommand;
      L     'c';
      ==I;
      L     50;	//Lenght in byte
      JC    Sndx;
      L     #tmpCommand;
      L     'g';
      ==I;
      L     8;	//Lenght in byte
      JC    Sndx;
      JU    SndA;
Sndx: T     DBW 86;	//COM.Telegram.LenAnswer
      JU    STOR;
SndA: NOP   0;
//Send O
      L     #tmpCommand;
      L     'O';
      <>I;
      JC    SndQ;
      L     #InStartValue;
      JU    Sd16;
//Send Q
SndQ: L     #tmpCommand;
      L     'Q';
      <>I;
      JC    SndT;
      L     #InFlowrateProduct;
      JU    Sd16;
//Send T
SndT: L     #tmpCommand;
      L     'T';
      <>I;
      JC    SndU;
      L     #InTargetValue;
      JU    Sd16;
//Send U
SndU: L     #tmpCommand;
      L     'U';
      <>I;
      JC    SndF;
      L     #InLimitPos;
      L     1000;
      *I;
      L     #InLimitNeg;
      +D;
      JU    Sd16;
//Send F
SndF: L     #tmpCommand;
      L     'F';
      <>I;
      JC    SndX;
      L     #InOffsetMoisture;
      JU    Sd16;
//Send X
SndX: L     #tmpCommand;
      L     'X';
      <>I;
      JC    SndR;
      L     #InDosingMax;
      JU    Sd16;
//Send R
SndR: L     #tmpCommand;
      L     'R';
      <>I;
      JC    SndS;
      L     #InProductGroup;
      T     DBD 36;	//COM.Element.InOutValue
      L     12;	//Convert DInt to 2-ASCII
      T     DBW 0;	//COM.CODE;
      L     2;	//Lenght in byte
      JU    Snd1;
//Send S
SndS: L     #tmpCommand;
      L     'S';
      <>I;
      JC    SndZ;
      LAR1  #tmpAddrOutStateTarget;
      L     B [AR1,P#1.0];
      T     DBD 36;	//COM.Element.InOutValue
      L     32;	//Convert Hex to 2-ASCII
      T     DBW 0;	//COM.CODE
      L     2;	//Lenght in byte
      JU    Snd1;
Sd16: T     DBD 36;	//COM.Element.InOutValue
      L     16;	//Convert DInt to 6-ASCII
      T     DBW 0;	//COM.CODE
      L     6;	//Lenght in Byte
Snd1: T     DBW 78;	//COM.Telegram.Len
      CDB;	//ComDB->Instanz-DB
      UC    "GCS7_RS485Ctrl";	//Convert (CODE=DBW0)
      CDB;	//ElementDB->Instanz-DB
SndZ: JU    STOR;
//--- Get done ---------------
//Copy reveived data to element
Rcv:  R     #OutComFault;
      L     #tmpCommand;
      L     'c';
      <>I;
      JC    Rcvg;
      R     #Par.OutStateTarget.ClearPowerFlag;
//Nominal target value
      L     0;	//Character offset
      T     DBW 40;	//COM.Element.AddrOffset
      L     26;	//Convert 6-ASCII to DInt
      T     DBW 0;	//COM.CODE
      CDB;	//ComDB->Instanz-DB
      UC    "GCS7_RS485Ctrl";	//Convert (CODE=DBW0)
      CDB;	//ElementDB->Instanz-DB
      L     DBD 36;	//COM.Element.InOutValue
      T     #OutTargetValue;
//Actual value
      L     6;	//Character offset
      T     DBW 40;	//COM.Element.AddrOffset
      L     26;	//Convert 6-ASCII to DInt
      T     DBW 0;	//COM.CODE
      CDB;	//ComDB->Instanz-DB
      UC    "GCS7_RS485Ctrl";	//Convert (CODE=DBW0)
      CDB;	//ElementDB->Instanz-DB
      L     DBD 36;	//COM.Element.InOutValue
      T     #OutActualValue;
//Product flowrate
      L     12;	//Character offset
      T     DBW 40;	//COM.Element.AddrOffset
      L     26;	//Convert 6-ASCII to DInt
      T     DBW 0;	//COM.CODE
      CDB;	//ComDB->Instanz-DB
      UC    "GCS7_RS485Ctrl";	//Convert (CODE=DBW0)
      CDB;	//ElementDB->Instanz-DB
      L     DBD 36;	//COM.Element.InOutValue
      T     #OutFlowrateProduct;
//Total product flowrate
      L     18;	//Character offset
      T     DBW 40;	//COM.Element.AddrOffset
      L     28;	//Convert 8-ASCII to DInt
      T     DBW 0;	//COM.CODE
      CDB;	//ComDB->Instanz-DB
      UC    "GCS7_RS485Ctrl";	//Convert (CODE=DBW0)
      CDB;	//ElementDB->Instanz-DB
      A     #CmdNewJob;	//[4.1]
      JC    rcJ1;	//[4.1]
      L     DBD 36;	//COM.Element.InOutValue
      T     #OutTotalProduct;
//Target value MOZE
rcJ1: L     26;	//Character offset
      T     DBW 40;	//COM.Element.AddrOffset
      L     26;	//Convert 6-ASCII to DInt
      T     DBW 0;	//COM.CODE
      CDB;	//ComDB->Instanz-DB
      UC    "GCS7_RS485Ctrl";	//Convert (CODE=DBW0)
      CDB;	//ElementDB->Instanz-DB
      L     DBD 36;	//COM.Element.InOutValue
      T     #OutFlowrateWaterTarget;
//Actual value MOZE
      L     32;	//Character offset
      T     DBW 40;	//COM.Element.AddrOffset
      L     26;	//Convert 6-ASCII to DInt
      T     DBW 0;	//COM.CODE
      CDB;	//ComDB->Instanz-DB
      UC    "GCS7_RS485Ctrl";	//Convert (CODE=DBW0)
      CDB;	//ElementDB->Instanz-DB
      L     DBD 36;	//COM.Element.InOutValue
      T     #OutFlowrateWater;
//Total water
      L     38;	//Character offset
      T     DBW 40;	//COM.Element.AddrOffset
      L     28;	//Convert 8-ASCII to DInt
      T     DBW 0;	//COM.CODE
      CDB;	//ComDB->Instanz-DB
      UC    "GCS7_RS485Ctrl";	//Convert (CODE=DBW0)
      CDB;	//ElementDB->Instanz-DB
      A     #CmdNewJob;	//[4.1]
      JC    rcJ2;	//[4.1]
      L     DBD 36;	//COM.Element.InOutValue
      T     #OutTotalWater;
//LC status
rcJ2: L     46;	//Character offset
      T     DBW 40;	//COM.Element.AddrOffset
      L     42;	//Convert 2-ASCII to Hex
      T     DBW 0;	//COM.CODE
      CDB;	//ComDB->Instanz-DB
      UC    "GCS7_RS485Ctrl";	//Convert (CODE=DBW0)
      CDB;	//ElementDB->Instanz-DB
      L     DBD 36;	//COM.Element.InOutValue
      LAR1  #tmpAddrOutLCState;
      T     B [AR1,P#1.0];	//-->#OutLCState
//Alarm number
      L     48;	//Character offset
      T     DBW 40;	//COM.Element.AddrOffset
      L     22;	//Convert 2-ASCII to DInt
      T     DBW 0;	//COM.CODE
      CDB;	//ComDB->Instanz-DB
      UC    "GCS7_RS485Ctrl";	//Convert (CODE=DBW0)
      CDB;	//ElementDB->Instanz-DB
      L     DBD 36;	//COM.Element.InOutValue
      T     #OutAlarmNr;
      L     1;
      SLD;
      SRD   1;	//Clear Alarm Bit 0
      SLD   1;
      CAD;	//Replace akku to correct bit order
      LAR1  #tmpAddrOutLCAlarm;
      T     D [AR1,P#0.0];	//#OutLCAlarm
      JU    STOR;
//-- Not erasable weight --- 
Rcvg: L     #tmpCommand;
      L     'g';
      <>I;
      JC    RcvS;
//Not erasable total of MOZE
      L     0;	//Character offset
      T     DBW 40;	//COM.Element.AddrOffset
      L     28;	//Convert 8-ASCII to DInt
      T     DBW 0;	//COM.CODE
      CDB;	//ComDB->Instanz-DB
      UC    "GCS7_RS485Ctrl";	//Convert (CODE=DBW0)
      CDB;	//ElementDB->Instanz-DB
      L     DBD 36;	//COM.Element.InOutValue
      T     #OutNotErasableWater;
      JU    STOR;
//--- Put done ---------------
RcvS: L     #tmpCommand;
      L     'S';
      <>I;
      JC    RcvX;
      A     #Par.OutStateTarget.AlarmReset;
      R     #CmdFaultReset;
      S     #OutFaultResetDone;
      AN    #Par.OutStateTarget.ClearLoopDatas;
      JC    STOR;
      R     #Par.OutStateTarget.ClearLoopDatas;
      R     #CmdNewJob;
      L     0;	//Clear
      T     #OutTotalProduct;	// -> Total of product flowrate
      T     #OutTotalWater;	// -> Total of dosing water
RcvX: JU    STOR;
NETWORK
TITLE = PC Control
//=== Test Object number =====================
PC:   L     "SYS_DirectCtrlDB".PC.ObjectNo;	//PCControl.ObjectNo
      L     #Par.ParObjectNo;	//Input ObjectNo
      <>I;
      JC    Ctrl;
//=== Test OType      ========================
      L     1023;	//Input object type
      L     "SYS_DirectCtrlDB".PC.ObjectType;	//PCControl.ObjectType
      <>I;
      JC    Ctrl;
//=== Test Handshake =========================
      A     "SYS_DirectCtrlDB".PC.Hsk.FExamine;	//Handshake.FExamine
      JC    pExa;
      A     "SYS_DirectCtrlDB".PC.Hsk.FDefineCmd;	//Handshake.FDefineCmd
      JC    pCmd;
      A     "SYS_DirectCtrlDB".PC.Hsk.FDefinePara;	//Handshake.FDefinePara
      JC    pPar;
pIni: L     2;	//FcInit
      UC    "SYS_DirectCtrl";
      JU    Ctrl;
//Write parameter 
pPar: NOP   0;
//Write new commands from PC to Interface of group 
pCmd: A     "SYS_DirectCtrlDB".PC.Cmd1[1];	//Cmd1[1]  =CmdLimitOn
      S     #InLimitOn;
      A     "SYS_DirectCtrlDB".PC.Cmd2[1];	//Cmd2[1]  =CmdLimitOff
      R     #InLimitOn;
      A     "SYS_DirectCtrlDB".PC.Cmd1[4];	//Cmd1[4]  =CmdNewValue
      S     #CmdNewValue;
      A     "SYS_DirectCtrlDB".PC.Cmd1[5];	//Cmd1[5]  =CmdNewJob
      S     #CmdNewJob;
      A     "SYS_DirectCtrlDB".PC.Cmd1[11];	//Cmd1[11] =CmdFaultReset
      S     #CmdFaultReset;
      A     "SYS_DirectCtrlDB".PC.Cmd1[13];	//Cmd1[13] =CmdManualOn
      S     #InManual;
      A     "SYS_DirectCtrlDB".PC.Cmd2[13];	//Cmd2[13] =CmdManualOff
      R     #InManual;
//Define Value
      AN    "SYS_DirectCtrlDB".PC.Hsk.FDefineValue;	// PC.Hsk.FDefineValue
      ON    #InManual;
      JC    pIni;
      LAR1  P#DBX 58.0;
      L     DBD [AR1,P#6.0];
      T     #InStartValue;
      L     DBD [AR1,P#10.0];
      T     #InFlowrateProduct;
      L     DBD [AR1,P#14.0];
      T     #InTargetValue;
      L     DBW [AR1,P#18.0];
      T     #InLimitPos;
      L     DBW [AR1,P#20.0];
      T     #InLimitNeg;
      L     DBD [AR1,P#22.0];
      T     #InOffsetMoisture;
      L     DBD [AR1,P#26.0];
      T     #InDosingMax;
      L     DBW [AR1,P#30.0];
      T     #InProductGroup;
      JU    pIni;
pExa: TAR2;	//Address dynamic datas
      T     "SYS_DirectCtrlDB".GC.InDynAddr;	//-->PCControl.GC.InDynAddr
      L     #tmpLenDyn;	//Length dynamic datas
      T     "SYS_DirectCtrlDB".GC.InDynLen;	//-->PCControl.GC.InDynLen
      L     0;
      T     "SYS_DirectCtrlDB".GC.InParaAddr;	//-->PCControl.GC.InParaAddr
      T     "SYS_DirectCtrlDB".GC.InParaLen;	//-->PCControl.GC.InParaLen
      L     1;	//Code FcExamine
      UC    "SYS_DirectCtrl";
      L     10;	//Revision
      T     "SYS_DirectCtrlDB".GC.Revision;
Ctrl: NOP   0;
NETWORK
TITLE = [5.0] LCParameter
      L     #Par.ParObjectNo;
      L     "SYS_DirectCtrlLCDB".PC.ObjectNo;
      <>I;
      JC    LCP0;
      T     "SYS_DirectCtrlLCDB".GC.InObjectNo;
      L     #Par.ParComDB;
      T     "SYS_DirectCtrlLCDB".GC.InDBNr;
      L     #Par.ParLCAddr;
      T     "SYS_DirectCtrlLCDB".GC.InLCAddr;
LCP0: NOP   0;
NETWORK
TITLE =  Read LC data
      OPN   DB [#tmpComDB];
      L     #Par.ParLCIdx;
      T     DBW 34;	//COM.Element.Index;
      L     1;	//Read LC data
      T     DBW 0;	//COM.CODE;
      CDB;
      UC    "GCS7_RS485Ctrl";
      CDB;
      L     #tmpFBNO;
      T     DBW 52;	//COM.LC0.FBNO;   
      L     DINO;
      T     DBW 54;	//COM.LC0.DINO;
      TAR2  DBD 56;	//COM.LC0.AddrDyn;        
      L     0;
      T     DBD 60;	//COM.LC0.AddrPara;       
      L     #Par.ParLCAddr;
      T     DBD 64;	//COM.Telegram.LCAddr;
NETWORK
TITLE =  All State Init
//===Clear tmp Variable
      SET;
      R     #tmpClearCmdFlag;
//===Global Group Orders===
      A     #InLocal;
      AN    #InManual;
      O     #InHWStop;
      O     #InDPFault;
      =     #tmpLocal;
//---FaultReset is on---
      A     "GCS7_Gr_OutFaultReset";	//Gr.OutFaultReset
      S     #CmdFaultReset;
//--- tmpFault   
      LAR1  #tmpAddrOutLCAlarm;
      L     D [AR1,P#0.0];	//#OutLCAlarm
      LAR1  #tmpAddrParFilter;
      L     D [AR1,P#0.0];	//#Par.ParFilter;
      INVD;	//Invers filter mask
      AD;
      L     0;
      <>D;
      O(;
      L     #OutAlarmNr;
      L     17;	//---Exception faults
      >I;
      );
      =     #tmpFault;
      A     #InpGroupAlarm;	//---Fault with InpGroupAlarm
      O     #InpProductAlarm;	//---Fault with InpProductAlarm
      A     #tmpFault;
      O     #OutComFault;	//---Communication fault
      =     #tmpFault;
      A     DBX 50.0;	//COM.LC0.CmdPut
      O     DBX 50.1;	//COM.LC0.CmdGet
      =     #tmpComActive;
//---CmdNewJob sets CmdNewValue
      A     #CmdNewJob;
      S     #CmdNewValue;
      AN    #CmdNewJob;	//[4.1]
      JC    NJJ0;	//[4.1]
      L     0;	//[4.1]Clear
      T     #OutTotalProduct;	//[4.1] -> Total of product flowrate
      T     #OutTotalWater;	//[4.1] -> Total of dosing water
NJJ0: NOP   0;	//[4.1]
//---LC State target commands
      A     #InLimitOn;	//Set limit active...
      XN    #Par.OutStateTarget.LimitActive;	// ..if both signals are different
      AN    #CmdFaultReset;
      AN    #CmdNewJob;
      O     #tmpComActive;
      O     #OutRequestActive;
      O     #OutComFault;
      JC    nVal;
      A     #CmdFaultReset;
      =     #Par.OutStateTarget.AlarmReset;
      =     #Par.OutStateTarget.ClearPowerFlag;
      A     #InLimitOn;
      =     #Par.OutStateTarget.LimitActive;
      A     #CmdNewJob;
      =     #Par.OutStateTarget.ClearLoopDatas;
      JU    CmdS;
//--- New Value
nVal: AN    #CmdNewValue;
      R     #OutNewValueActive;
      JC    nReq;
      A     #tmpComActive;
      O     #OutComFault;
      O     #OutRequestActive;
      ON    #StOk;
      JC    nReq;
      AN    #Par.OutComFlags.O_Done;
      AN    #Par.ParComFlags.Without_O;
      JC    CmdO;
      AN    #Par.OutComFlags.Q_Done;
      AN    #Par.ParComFlags.Without_Q;
      JC    CmdQ;
      AN    #Par.OutComFlags.T_Done;
      AN    #Par.ParComFlags.Without_T;
      JC    CmdT;
      AN    #Par.OutComFlags.U_Done;
      AN    #Par.ParComFlags.Without_U;
      JC    CmdU;
      AN    #Par.OutComFlags.F_Done;
      AN    #Par.ParComFlags.Without_F;
      JC    CmdF;
      AN    #Par.OutComFlags.X_Done;
      AN    #Par.ParComFlags.Without_X;
      JC    CmdX;
      AN    #Par.OutComFlags.R_Done;
      AN    #Par.ParComFlags.Without_R;
      JC    CmdR;
      R     #OutNewValueActive;
      R     #CmdNewValue;
      S     #tmpClearCmdFlag;
//---New Request
nReq: A     #tmpComActive;
      JC    STAT;
      S     #OutRequestActive;
      AN    #Par.OutComFlags.c_Done;
      JC    Cmdc;
      AN    #Par.OutComFlags.g_Done;
      JC    Cmdg;
      S     #tmpClearCmdFlag;
      R     #OutRequestActive;
      JU    OUT;
NETWORK
TITLE = States
//===State machine===
STAT: A     #StOk;
      JC    S2;
      A     #StFault;
      JC    S4;
      A     #StFalse;
      JC    S5;
      S     #StOk;	//Init
NETWORK
TITLE =  StOk
xS2:  S     #StOk;
      R     #StFalse;
      R     #StFault;
      R     #CmdFaultReset;
      R     #OutFaultResetDone;
      L     B#(3, 4);	//Message Operator ('fault cancelled' )
      JU    LOG;
S2:   A     #tmpFault;	//Condition for StFault/StFalse
      AN    #tmpLocal;
      JC    xS45;	//StXxx -> StFault transition flag
      A     #tmpFault;	//Condition for StFault/StFalse
      S     #StFalse;
      R     #StOk;
      JU    OUT;
NETWORK
TITLE =  StFault
S4:   AN    #tmpFault;	//---Condition for StOk
      A     #CmdFaultReset;
      JC    xS2;
      A     #tmpLocal;	//---Condition for StFalse
      JC    xS45;
      A     #OutFaultResetDone;	//reLOG fault
      JC    xS45;
      JU    OUT;
NETWORK
TITLE =  StFalse
//Automatic fault reset
S5:   AN    #tmpFault;	//---Condition for StOk
      JC    xS2;
      AN    #tmpLocal;	//---Condition for StFault
      JC    xS45;	//StXxx -> StFault transition flag
      A     #OutFaultResetDone;	//---Fault reset
      S     #CmdFaultReset;
      R     #OutFaultResetDone;
      JU    OUT;
NETWORK
TITLE = Communication start
Cmdc: S     #Par.OutComFlags.c_Done;
      L     'c';
      JU    GET;
Cmdg: S     #Par.OutComFlags.g_Done;
      L     'g';
      JU    GET;
CmdO: A     #Par.ParComFlags.Without_O;
      JC    OUT;
      S     #Par.OutComFlags.O_Done;
      S     #OutNewValueActive;
      L     'O';
      JU    PUT;
CmdQ: A     #Par.ParComFlags.Without_Q;
      JC    OUT;
      S     #Par.OutComFlags.Q_Done;
      S     #OutNewValueActive;
      L     'Q';
      JU    PUT;
CmdT: A     #Par.ParComFlags.Without_T;
      JC    OUT;
      S     #Par.OutComFlags.T_Done;
      S     #OutNewValueActive;
      L     'T';
      JU    PUT;
CmdU: A     #Par.ParComFlags.Without_U;
      JC    OUT;
      S     #Par.OutComFlags.U_Done;
      S     #OutNewValueActive;
      L     'U';
      JU    PUT;
CmdF: A     #Par.ParComFlags.Without_F;
      JC    OUT;
      S     #Par.OutComFlags.F_Done;
      S     #OutNewValueActive;
      L     'F';
      JU    PUT;
CmdX: A     #Par.ParComFlags.Without_X;
      JC    OUT;
      S     #Par.OutComFlags.X_Done;
      S     #OutNewValueActive;
      L     'X';
      JU    PUT;
CmdR: A     #Par.ParComFlags.Without_R;
      JC    OUT;
      S     #Par.OutComFlags.R_Done;
      S     #OutNewValueActive;
      L     'R';
      JU    PUT;
CmdS: L     'S';
      JU    PUT;
PUT:  SET;
      S     DBX 50.0;	//COM.LC0.CmdPut ;
      JU    ALL1;
GET:  SET;
      S     DBX 50.1;	//COM.LC0.CmdGet ;
ALL1: S     #tmpComActive;
      T     DBB 51;	//COM.LC0.Command;
      JU    OUT;
NETWORK
TITLE = LOG
xS45: S     #tmpClearCmdFlag;	//to clear x_done flags
      R     #StOk;
      R     #OutFaultResetDone;
      R     #OutRequestActive;
      A     #InLocal;	//---InLocal=1 -> StFalse -> no LOG message
      AN    #InManual;
      S     #StFalse;
      R     #StFault;
      JC    OUT;
      A     #StFault;	// 2.1: Fault flag only when transition -> StFault
      JC    S4J2;
      S     "GCS7_Gr_InFaultFlag";	// 2.1: Gr.InFaultFlag
      CALL  "SYS_Horn_Code" (
           FcCode                   := 1,
           ParObjectType            := 1023,
           ParObjectNo              := #Par.ParObjectNo,
           ParHornCode              := #Par.ParHornCode);
S4J2: SET;	// 2.1:
      S     #StFault;
      R     #StFalse;
      L     B#(1, 14);
      A     #OutComFault;
      JC    LOG;
      L     B#(1, 1);
      A     #Par.OutLCAlarm.SoftwareTimerOverflow;
      JC    LOG;
      L     B#(1, 2);
      A     #Par.OutLCAlarm.PosLimitBand;
      JC    LOG;
      L     B#(1, 3);
      A     #Par.OutLCAlarm.NegLimitBand;
      JC    LOG;
      L     B#(1, 5);
      A     #Par.OutLCAlarm.MOZEFncAlarm;
      JC    LOG;
      L     B#(1, 6);
      A     #Par.OutLCAlarm.MOZEComAlarm;
      JC    LOG;
      L     B#(1, 7);
      A     #Par.OutLCAlarm.MOZEConfigAlarm;
      JC    LOG;
      L     B#(1, 8);
      A     #Par.OutLCAlarm.MOZEMinSetPointAlarm;
      JC    LOG;
      L     B#(1, 9);
      A     #Par.OutLCAlarm.MOZEMaxSetPointAlarm;
      JC    LOG;
      L     B#(1, 10);
      A     #Par.OutLCAlarm.MYFBFncAlarm;
      JC    LOG;
      L     B#(1, 11);
      A     #Par.OutLCAlarm.MYFBComAlarm;
      JC    LOG;
      L     B#(1, 12);
      A     #Par.OutLCAlarm.MYFBConfigAlarm;
      JC    LOG;
      L     B#(1, 13);
      A     #Par.OutLCAlarm.MYFBMeasureAlarm;
      JC    LOG;
      L     B#(1, 15);
      A     #Par.OutLCAlarm.FlowFncAlarm;
      JC    LOG;
      L     B#(1, 16);
      A     #Par.OutLCAlarm.FlowComAlarm;
      JC    LOG;
      L     B#(1, 17);
      A     #Par.OutLCAlarm.FlowConfigAlarm;
      JC    LOG;
      L     B#(1, 14);	//COM communication
      JU    LOG;
LOG:  A     #Par.ParLogOff;	//---Set LOG Message
      JC    SAVE;
      T     #tmpLOGvalue;
      L     W#16#FF;
      AW;
      T     #OutAlarmNrLog;
      CALL  "GCS7_LogConvert" (
           ObjectNo                 := #Par.ParObjectNo,
           MsgType                  := #Par.ParMsgType,
           ClassMsgTxt              := #tmpLOGvalue,
           OType                    := 1023);	//LOG Message Converter / Entry / Contains Class and TextNo
NETWORK
TITLE = Global End
OUT:  NOP   0;
SAVE: SET;	//---Clear all commands
      AN    #tmpClearCmdFlag;	//---Clear command flags (x_done)
      JC    STC0;
      R     #Par.OutComFlags.c_Done;
      R     #Par.OutComFlags.g_Done;
      R     #Par.OutComFlags.O_Done;
      R     #Par.OutComFlags.Q_Done;
      R     #Par.OutComFlags.T_Done;
      R     #Par.OutComFlags.U_Done;
      R     #Par.OutComFlags.F_Done;
      R     #Par.OutComFlags.X_Done;
      R     #Par.OutComFlags.R_Done;
//--Output for group 
STC0: AN    #InLocal;
      A     #InDPFault;
      S     "GCS7_Gr_InDPFault";
      AN    #InLocal;
      A     #InHWStop;
      S     "GCS7_Gr_InHWStop";
NETWORK
TITLE = State Code
      L     3;	//Code: ok
      A     #StOk;
      JC    STC;
      L     45;	//Code: false HWStop
      A     #StFalse;
      A     #InHWStop;
      JC    STC;
      L     55;	//Code: false DPFault
      A     #StFalse;
      A     #InDPFault;
      JC    STC;
      L     5;	//Code: false
      A     #StFalse;
      JC    STC;
      L     32;	//Code: fault
STC:  L     #StCode;	//Old state code
      TAK;
      T     #StCode;	//Save state code
      <>I;
      L     3;	//Load code for CBit methode
      CC    "SYS_CBitCtrl";
NETWORK
TITLE =  Store LC data
      L     #Par.ParLCIdx;
      T     DBW 34;	//COM.Element.Index; 
      L     2;	//Store LC data
      T     DBW 0;	//COM.CODE;
      CDB;
      UC    "GCS7_RS485Ctrl";
      CDB;
NETWORK
TITLE = Restore 
STOR: NOP   0;
END_FUNCTION_BLOCK

FUNCTION_BLOCK "GCS7_E_MOZE"	// FB 24
TITLE = MOZE Liquids Flow Control
//  
//COPYRIGHT:    (C) 1997  BUHLER AG, CH-9240 UZWIL, SWITZERLAND
//
//PRODUCT:      GCS7
//
//TITLE:        Element MOZE Liquids Flow Control
//
//-------------------------------------------------------------------------
//
//IDENT:        AUTHOR:             DEPT:                      DATE:
//
//FB24.5.0      A.Egli              CT3                        05-Jan-2005
//              Parameter Upload (uses DB10)
//FB24.4.0      A. Egli             CT3                        17-Jun-2002
//              New Release with one block 
//FB24.2.2      A. Egli             CT3                        17-Mar-2000
//              Length for answer telegram
//FB24.2.1      S. Kalberer         CT3                        06-Dec-1999
//              No horn if InLocal
//FB24.2A       A. Egli             CT3                        04-Mai-1998
//              StFault = StCode 32
//FB24.1B       A. Egli             CT3                        16-Apr-1998
//              Test
//FB24.1A       S. Kalberer         AEE61                      15-Aug-1997
//              1st Release in S7
//
//-------------------------------------------------------------------------
//
//PURPOSE:      MANUAL : see [LFCxxMAN]
//
//RESTRICTIONS: S7
//              ACCU2: Pointer to dynamic datas of the element
//              ACCU1: Pointer to parameter datas of the element
//
//-------------------------------------------------------------------------
//=======================================================
//Log Message: 
//------------------------------------------------------
//  1  ext 5 VDC not available     = #OutLCAlarm.Ext5NotAvailable
//  2  ext 24 VDC not available    = #OutLCAlarm.Ext24NotAvailable
//  3  overload of an output       = #OutLCAlarm.OverloadOutput
//  4  overload output operation   = #OutLCAlarm.OverloadOutputOper
//  5  turbine flowmeter faulty    = #OutLCAlarm.TurbineFlowFaulty
//  6  turbine flowmeter 1 faulty  = #OutLCAlarm.TurbineFlow1Faulty
//  7  alarm during closing        = #OutLCAlarm.AlarmClosing
//  8  alarm during opening        = #OutLCAlarm.AlarmOpening
//  9  no valid nominal value      = #OutLCAlarm.NoValidNominalValue
//  10 AD alarm                    = #OutLCAlarm.ADAlarm
//  11 invalid nominal value       = #OutLCAlarm.InvalidNominalValue
//  13 fault cancelled
//  14 fault communication         = OutComFault
//  15 exception error
//  16 stopped
//  17 started
//
//=======================================================
//StCode:  State               
//------------------------------------------------------
//32   StFault                 
// 1   StStopped                      Stopped
//41   Stopped.HWStop                 StStopped + InHWStop 
//51   Stopped.DPFault                StStopped + DPFault
// 3   StStarted               
// 5   StFalse                 
//
AUTHOR : EA
FAMILY : GCS7LL
NAME : MOZE
VERSION : 5.0
VAR
  StCode : INT ;	//Element state code
  InEnable : BOOL ;	//Enable to run the element (manual and automatic mode)
  spare0201 : BOOL ;
  spare0202 : BOOL ;
  spare0203 : BOOL ;
  CmdNewValue : BOOL ;	//Send new target values
  CmdNewJob : BOOL ;	//Clear actual values
  spare0206 : BOOL ;	//DI product alarm
  spare0207 : BOOL ;	//DI group alarm
  CmdOff : BOOL ;	//Pulse to stop the element (manual mode)
  CmdOn : BOOL ;	//Pulse to start the element (manual mode)
  CmdNext : BOOL ;	//Pulse to start the element in automatic mode
  CmdFaultReset : BOOL ;	//Command to reset fault
  InLocal : BOOL ;	//1= Local mode (no fault by start with service switch)
  InManual : BOOL ;	//1= Manual / 0= Automatic
  InReport : BOOL ;	//Report of all state transitions
  spare0307 : BOOL ;
  InHWStop : BOOL ;	//HW stop is detected, no fault
  InDPFault : BOOL ;	//DP-Fault is detected, no fault
  OutComFault : BOOL ;	//Communication fault
  spare0401 : BOOL ;
  OutRequestActive : BOOL ;	//Aux. signal request active
  OutFaultResetDone : BOOL ;	//Aux. signal fault reset done
  spare0406 : BOOL ;
  OutpDosingEnable : BOOL ;	//DO dosing enable
  StStopped : BOOL ;	//Element is stopped
  spare0501 : BOOL ;
  StStarted : BOOL ;	//Element is started
  spare0503 : BOOL ;
  StFault : BOOL ;	//Element has a communication or device fault
  StFalse : BOOL ;	//Element is in local mode and has a fault
  InFlowrateWater : DINT ;	//Is send to LC [0.1 l/h]
  InMinFlowrate : DINT ;	//Is send to LC [0.1 l/h]
  InMaxFlowrate : DINT ;	//Is send to LC [0.1 l/h]
  InNoOfValuesAverage : INT  := 1;	//Is send to LC [1..30]
  InVolumePerImpulse : INT ;	//Is send to LC [0.1 l]
  OutAlarmNr : INT ;	//Is read from LC [0..99]
  OutFlowrateWater : DINT ;	//Is read from LC [0.1 l/h]
  OutNotErasableWater : DINT ;	//Is read from LC (sum2) [0.1 l]
  OutTotalWater : DINT ;	//Is calulated by element
  OutAlarmNrLog : INT ;	//Last textnumber send to log
  Par : STRUCT
   ParObjectNo : INT ;	//Is used for communication with PC, e.g. for message
   ParMsgType : INT ;	//Is used for message (translation of state)
   ParHornCode : INT ;	//Is used by horn module
   ParLogOff : BOOL ;	//Report is off
   ParFilter : STRUCT 	//Filter to alarm 1=Ignore alarm
    spare00 : BOOL ;
    Ext5NotAvailable : BOOL ;	//Ext  5 VDC not available
    Ext24NotAvailable : BOOL ;	//Ext 24 VDC not available
    OverloadOutput : BOOL ;	//Overload of an output
    OverloadOutputOper : BOOL ;	//Overload output operation
    TurbineFlowFaulty : BOOL ;	//Turbine flowmeter faulty
    TurbineFlow1Faulty : BOOL ;	//Turbine flowmeter 1 faulty
    AlarmClosing : BOOL ;	//Alarm during closing
    AlarmOpening : BOOL ;	//Alarm during opening
    NoValidNominalValue : BOOL ;	//No valid nominal value
    ADAlarm : BOOL ;	//AD converter alarm
    InvalidNominalValue : BOOL ;	//Invalid nominal value
   END_STRUCT ;
   ParComFlags : STRUCT
    spare00 : BYTE ;
    Without_Q : BOOL ;	//Nominal output
    Without_N : BOOL ;	//Minimum nominal output
    Without_X : BOOL ;	//Maximum nominal output
    Without_D : BOOL ;	//Number of values to be averaged
    Without_G : BOOL ;	//Volume per impulse
    spare15 : BOOL ;
    spare16 : BOOL ;
    spare17 : BOOL ;
   END_STRUCT ;
   ParComDB : INT ;	//Communication DB
   ParLCIdx : INT ;	//Index of data record
   ParLCAddr : INT ;	//Address of LC
   OutLCState : STRUCT 	//Is read from LC
    spare00 : BYTE ;
    HostActive : BOOL ;	//Host control active
    DosingRelease : BOOL ;	//Dosing release
    AlarmActive : BOOL ;	//Alarm active
    spare13 : BOOL ;
    PowerFailure : BOOL ;	//Power failure
    OperationMessage : BOOL ;	//Operation message
    NominalValueReached : BOOL ;	//Nominal value reached
    DosingRunning : BOOL ;	//Dosing is running
   END_STRUCT ;
   OutLCAlarm : STRUCT 	//Alarm bit mask of OutAlarmNumber
    spare00 : BOOL ;
    Ext5NotAvailable : BOOL ;	//Ext  5 VDC not available
    Ext24NotAvailable : BOOL ;	//Ext 24 VDC not available
    OverloadOutput : BOOL ;	//Overload of an output
    OverloadOutputOper : BOOL ;	//Overload output operation
    TurbineFlowFaulty : BOOL ;	//Turbine flowmeter faulty
    TurbineFlow1Faulty : BOOL ;	//Turbine flowmeter 1 faulty
    AlarmClosing : BOOL ;	//Alarm during closing
    AlarmOpening : BOOL ;	//Alarm during opening
    NoValidNominalValue : BOOL ;	//No valid nominal value
    ADAlarm : BOOL ;	//AD Alarm
    InvalidNominalValue : BOOL ;	//Invalid nominal value
    spare14 : BOOL ;
    spare15 : BOOL ;
    spare16 : BOOL ;
    spare17 : BOOL ;
   END_STRUCT ;
   OutStateTarget : STRUCT 	//Command for LC, is send to LC
    spare00 : BYTE ;
    spare10 : BOOL ;
    spare11 : BOOL ;
    AlarmReset : BOOL ;	//Alarm reset
    spare13 : BOOL ;
    ClearPowerFlag : BOOL ;	//Clear powerfailure flag
    SetDosingRelease : BOOL ;	//Set dosing release
    ClearErasableTotal : BOOL ;	//Clear erasable total
    spare17 : BOOL ;
   END_STRUCT ;
   OutComFlags : STRUCT 	//Flags for communication
    d_Done : BOOL ;	//Actual value block 2 done
    Q_Done : BOOL ;	//Nominal output
    N_Done : BOOL ;	//Minimum nominal output
    X_Done : BOOL ;	//Maximum nominal output
    D_Done1 : BOOL ;	//Number of values to be averaged
    G_Done : BOOL ;	//Volume per impulse
   END_STRUCT ;
  END_STRUCT ;
END_VAR
VAR_TEMP
  tmpAddrOffset : DWORD ;	//store the Instance Pointer
  tmpLOGvalue : WORD ;	//LOG value
  tmpCommand : INT ;
  tmpFBNO : INT ;	//Number of the actual FB
  tmpFault : BOOL ;
  tmpComActive : BOOL ;	//Put or get is in queue
  tmpClearCmdFlag : BOOL ;	//Clear pattern Commands
  tmpOff : BOOL ;
  tmpOn : BOOL ;
  tmpReport : BOOL ;
  tmpLenDyn : DINT ;
  tmpAddrParFilter : DWORD ;	//Pointer to ParFilter
  tmpAddrOutLCState : DWORD ;	//Pointer to OutLCState
  tmpAddrOutLCAlarm : DWORD ;	//Pointer to OutLCAlarm
  tmpAddrOutStateTarget : DWORD ;	//Pointer to OutLCStateTarget
  tmpWt : DINT ;
  tmpComDB : INT ;
  tmpLocal : BOOL ;
  tmpLocalFault : BOOL ;
END_VAR
BEGIN
NETWORK
TITLE =  Start Global
      L     24;
      T     #tmpFBNO;
      L     64;
      T     #tmpLenDyn;	//--> Len dynamic data in byte
      TAR2;
      L     DW#16#FFFFFF;
      AD;
      T     #tmpAddrOffset;	//-->Addr Para
      L     P##Par;
      L     #tmpAddrOffset;
      +D;
      LAR1;
      L     P#8.0;	// P##ParFilter
      +D;
      T     #tmpAddrParFilter;	//-->Pointer to ParFilter
      TAR1;
      L     P#18.0;	//P##Par.OutLCState
      +D;
      T     #tmpAddrOutLCState;	//-->Pointer to OutLCState
      TAR1;
      L     P#20.0;	//P##Par.OutLCAlarm
      +D;
      T     #tmpAddrOutLCAlarm;	//-->Pointer to OutLCAlarm
      TAR1;
      L     P#22.0;	//P##Par.OutStateTarget
      +D;
      T     #tmpAddrOutStateTarget;	//-->Pointer to OutStateTarget
      L     #Par.ParComDB;
      T     #tmpComDB;
NETWORK
TITLE =  Call back function
//*****This functions are called by FBxxx (COM) ******
      OPN   DB [#tmpComDB];
      L     0;
      L     DBW 32;	//COM.Element.CODE;
      ==I;
      JC    PC;
      L     DBB 76;	//COM.Telegram.Command;
      T     #tmpCommand;
      L     1;
      L     DBW 32;	//COM.Element.CODE;
      ==I;
      JC    Send;
      L     2;
      ==I;
      JC    Rcv;
      L     4;	//NAK
      L     DBW 32;	//COM.Element.CODE;
      ==I;
      S     #OutComFault;	//fault MYEB communication
      JU    STOR;
//Read telegram length
Send: L     #tmpCommand;
      L     'd';
      ==I;
      L     18;	//Lenght in byte
      JC    Sndx;
      JU    SndA;
Sndx: T     DBW 86;	//COM.Telegram.LenAnswer
      JU    STOR;
SndA: NOP   0;
//Send Q
      L     #tmpCommand;
      L     'Q';
      <>I;
      JC    SndN;
      L     #InFlowrateWater;
      JU    Sd16;
//Send N
SndN: L     #tmpCommand;
      L     'N';
      <>I;
      JC    SndX;
      L     #InMinFlowrate;
      JU    Sd16;
//Send X
SndX: L     #tmpCommand;
      L     'X';
      <>I;
      JC    SndD;
      L     #InMaxFlowrate;
      JU    Sd16;
//Send D
SndD: L     #tmpCommand;
      L     'D';
      <>I;
      JC    SndG;
      L     #InNoOfValuesAverage;
      JU    Sd14;
//Send G
SndG: L     #tmpCommand;
      L     'G';
      <>I;
      JC    SndS;
      L     #InVolumePerImpulse;
Sd14: T     DBD 36;	//COM.Element.InOutValue
      L     14;	//Convert Integer to 4-ASCII
      T     DBW 0;	//COM.CODE;
      L     4;	//Lenght in byte
      JU    Snd1;
//Send S
SndS: L     #tmpCommand;
      L     'S';
      <>I;
      JC    SndZ;
      LAR1  #tmpAddrOutStateTarget;
      L     B [AR1,P#1.0];
      T     DBD 36;	//COM.Element.InOutValue
      L     32;	//Convert Hex to 2-ASCII
      T     DBW 0;	//COM.CODE
      L     2;	//Lenght in byte
      JU    Snd1;
Sd16: T     DBD 36;	//COM.Element.InOutValue
      L     16;	//Convert DInt to 6-ASCII
      T     DBW 0;	//COM.CODE
      L     6;	//Lenght in byte
Snd1: T     DBW 78;	//COM.Telegram.Len
      CDB;	//ComDB->Instanz-DB
      UC    "GCS7_RS485Ctrl";	//Convert (CODE=DBW0)
      CDB;	//ElementDB->Instanz-DB
SndZ: JU    STOR;
//--- Get done ---------------
//Copy reveived data to element
Rcv:  R     #OutComFault;
      L     #tmpCommand;
      L     'd';
      <>I;
      JC    RcvS;
      R     #Par.OutStateTarget.ClearPowerFlag;
//LC status
      L     0;	//Character offset
      T     DBW 40;	//COM.Element.AddrOffset
      L     42;	//Convert 2-ASCII to Hex
      T     DBW 0;	//COM.CODE
      CDB;	//ComDB->Instanz-DB
      UC    "GCS7_RS485Ctrl";	//Convert (CODE=DBW0)
      CDB;	//ElementDB->Instanz-DB
      L     DBD 36;	//COM.Element.InOutValue
      LAR1  #tmpAddrOutLCState;
      T     B [AR1,P#1.0];	//-->#OutLCState
//Alarm number / LC alarm bit mask
      L     2;	//Character offset
      T     DBW 40;	//COM.Element.AddrOffset
      L     22;	//Convert 2-ASCII to DInt
      T     DBW 0;	//COM.CODE
      CDB;	//ComDB->Instanz-DB
      UC    "GCS7_RS485Ctrl";	//Convert (CODE=DBW0)
      CDB;	//ElementDB->Instanz-DB
      L     DBD 36;	//COM.Element.InOutValue
      T     #OutAlarmNr;
      L     1;
      SLD;
      SRD   1;	//Clear Alarm Bit 0
      SLD   1;
      CAW;	//Replace akku to correct bit order
      LAR1  #tmpAddrOutLCAlarm;
      T     W [AR1,P#0.0];	//#OutLCAlarm
//Acutal output
      L     4;	//Character offset
      T     DBW 40;	//COM.Element.AddrOffset
      L     26;	//Convert 6-ASCII to DInt
      T     DBW 0;	//COM.CODE
      CDB;	//ComDB->Instanz-DB
      UC    "GCS7_RS485Ctrl";	//Convert (CODE=DBW0)
      CDB;	//ElementDB->Instanz-DB
      L     DBD 36;	//COM.Element.InOutValue
      T     #OutFlowrateWater;
//Not erasable total
      L     10;	//Character offset
      T     DBW 40;	//COM.Element.AddrOffset
      L     28;	//Convert 8-ASCII to DInt
      T     DBW 0;	//COM.CODE
      CDB;	//ComDB->Instanz-DB
      UC    "GCS7_RS485Ctrl";	//Convert (CODE=DBW0)
      CDB;	//ElementDB->Instanz-DB
      L     DBD 36;	//ERH.Element.InOutValue
      T     #tmpWt;
//---  Init first, if old value < 0  ---
      L     #OutNotErasableWater;
      L     0;
      <D;
      JC    rgZ2;
//---  Calculate Weight ---
      L     #tmpWt;
      L     #OutNotErasableWater;
      -D;
      JM    rgZ1;
      JU    rgPo;
rgZ1: L     L#100000000;
      +D;
rgPo: L     10000;	// Maximum change by relaod software
      >D;
      JC    rgZ2;
      TAK;
      L     #OutTotalWater;
      +D;
      T     #OutTotalWater;	//--> Total weight
rgZ2: L     #tmpWt;
      T     #OutNotErasableWater;
      JU    STOR;
//--- Put done ---------------
RcvS: L     #tmpCommand;
      L     'S';
      <>I;
      JC    RcvX;
      A     #Par.OutStateTarget.AlarmReset;
      R     #CmdFaultReset;
      S     #OutFaultResetDone;
      AN    #Par.OutStateTarget.ClearErasableTotal;
      JC    STOR;
      R     #CmdNewJob;
RcvX: NOP   0;
STOR: BEU;
NETWORK
TITLE = PC Control
//=== Test Object number =====================
PC:   L     "SYS_DirectCtrlDB".PC.ObjectNo;	//PCControl.ObjectNo
      L     #Par.ParObjectNo;	//Input ObjectNo
      <>I;
      JC    Ctrl;
//=== Test OType      ========================
      L     1024;	//Input object type
      L     "SYS_DirectCtrlDB".PC.ObjectType;	//PCControl.ObjectType
      <>I;
      JC    Ctrl;
//=== Test Handshake =========================
      A     "SYS_DirectCtrlDB".PC.Hsk.FExamine;	//Handshake.FExamine
      JC    pExa;
      A     "SYS_DirectCtrlDB".PC.Hsk.FDefineCmd;	//Handshake.FDefineCmd
      JC    pCmd;
      A     "SYS_DirectCtrlDB".PC.Hsk.FDefinePara;	//Handshake.FDefinePara
      JC    pPar;
pIni: L     2;	//FcInit
      UC    "SYS_DirectCtrl";
      JU    Ctrl;
//Write parameter 
pPar: NOP   0;
//Write new commands from PC to Interface of group 
pCmd: A     "SYS_DirectCtrlDB".PC.Cmd1[4];	//Cmd1[4]  =CmdNewValue
      S     #CmdNewValue;
      A     "SYS_DirectCtrlDB".PC.Cmd1[5];	//Cmd1[5]  =CmdNewJob
      S     #CmdNewJob;
      A     "SYS_DirectCtrlDB".PC.Cmd1[8];	//Cmd1[8]  =CmdOff
      S     #CmdOff;
      A     "SYS_DirectCtrlDB".PC.Cmd1[9];	//Cmd1[9]  =CmdOn
      S     #CmdOn;
      A     "SYS_DirectCtrlDB".PC.Cmd1[10];	//Cmd1[10] =CmdNext
      S     #CmdNext;
      A     "SYS_DirectCtrlDB".PC.Cmd1[11];	//Cmd1[11] =CmdFaultReset
      S     #CmdFaultReset;
      A     "SYS_DirectCtrlDB".PC.Cmd1[13];	//Cmd1[13] =CmdManualOn
      S     #InManual;
      A     "SYS_DirectCtrlDB".PC.Cmd2[13];	//Cmd2[13] =CmdManualOff
      R     #InManual;
      A     "SYS_DirectCtrlDB".PC.Cmd1[14];	//Cmd1[14] =CmdReportOn
      S     #InReport;
      A     "SYS_DirectCtrlDB".PC.Cmd2[14];	//Cmd2[14] =CmdReportOff
      R     #InReport;
//Define Value
      AN    "SYS_DirectCtrlDB".PC.Hsk.FDefineValue;	// PC.Hsk.FDefineValue
      ON    #InManual;
      JC    pIni;
      LAR1  P#DBX 58.0;
      L     DBD [AR1,P#6.0];
      T     #InFlowrateWater;
      L     DBD [AR1,P#10.0];
      T     #InMinFlowrate;
      L     DBD [AR1,P#14.0];
      T     #InMaxFlowrate;
      L     DBW [AR1,P#18.0];
      T     #InNoOfValuesAverage;
      L     DBW [AR1,P#20.0];
      T     #InVolumePerImpulse;
      JU    pIni;
pExa: TAR2;	//Address dynamic datas
      T     "SYS_DirectCtrlDB".GC.InDynAddr;	//-->PCControl.GC.InDynAddr
      L     #tmpLenDyn;	//Length dynamic datas
      T     "SYS_DirectCtrlDB".GC.InDynLen;	//-->PCControl.GC.InDynLen
      L     0;
      T     "SYS_DirectCtrlDB".GC.InParaAddr;	//-->PCControl.GC.InParaAddr
      T     "SYS_DirectCtrlDB".GC.InParaLen;	//-->PCControl.GC.InParaLen
      L     1;	//Code FcExamine
      UC    "SYS_DirectCtrl";
      L     10;	//Revision
      T     "SYS_DirectCtrlDB".GC.Revision;
Ctrl: NOP   0;
NETWORK
TITLE = [5.0] LCParameter
      L     #Par.ParObjectNo;
      L     "SYS_DirectCtrlLCDB".PC.ObjectNo;
      <>I;
      JC    LCP0;
      T     "SYS_DirectCtrlLCDB".GC.InObjectNo;
      L     #Par.ParComDB;
      T     "SYS_DirectCtrlLCDB".GC.InDBNr;
      L     #Par.ParLCAddr;
      T     "SYS_DirectCtrlLCDB".GC.InLCAddr;
LCP0: NOP   0;
NETWORK
TITLE =  Read LC data
      OPN   DB [#tmpComDB];
      L     #Par.ParLCIdx;
      T     DBW 34;	//COM.Element.Index;
      L     1;	//Read LC data
      T     DBW 0;	//COM.CODE;
      CDB;
      UC    "GCS7_RS485Ctrl";
      CDB;
      L     #tmpFBNO;
      T     DBW 52;	//COM.LC0.FBNO;
      L     DINO;
      T     DBW 54;	//COM.LC0.DINO;
      TAR2  DBD 56;	//COM.LC0.AddrDyn;        
      L     #tmpAddrOffset;
      T     DBD 60;	//COM.LC0.AddrPara;       
      L     #Par.ParLCAddr;
      T     DBD 64;	//COM.Telegram.LCAddr;
NETWORK
TITLE =  All State Init
//===Clear tmp Variable
      SET;
      R     #tmpClearCmdFlag;
//===Global Group Orders===
      A     "GCS7_Gr_OutManualOn";	//Global.OutManualOn
      S     #InManual;
      A     "GCS7_Gr_OutManualOff";	//Global.OutManualOff
      R     #InManual;
      A     #InManual;
      S     "GCS7_Gr_InManual";	//Global.InManualMode
//---Report is on---
      O     "GCS7_Gr_OutReportAll";	//---Global OutReportAll
      O     #InReport;
      =     #tmpReport;
//---FaultReset is on---
      A     "GCS7_Gr_OutFaultReset";	//Gr.OutFaultReset
      S     #CmdFaultReset;
//---tmpLocal---
      A     #InLocal;
      AN    #InManual;
      =     #tmpLocalFault;
      A     #tmpLocalFault;
      O     #InHWStop;
      O     #InDPFault;
      =     #tmpLocal;
//---Off---
      AN    #InEnable;
      AN    #InManual;
      O     #tmpLocal;
      O     #CmdOff;
      =     #tmpOff;
//---On---
      O     #CmdNext;
      AN    #InManual;
      O     #CmdOn;
      AN    #tmpOff;
      =     #tmpOn;
//--- tmpFault   
      LAR1  #tmpAddrOutLCAlarm;
      L     W [AR1,P#0.0];	//#OutLCAlarm
      LAR1  #tmpAddrParFilter;
      L     W [AR1,P#0.0];	//#Par.ParFilter;
      INVI;	//Invers filter mask
      AW;
      L     0;
      <>I;
      O(;
      L     #OutAlarmNr;
      L     11;	//---Exception faults
      >I;
      );
      O     #OutComFault;	//---Communication fault
      =     #tmpFault;
      A     DBX 50.0;	//COM.LC0.CmdPut
      O     DBX 50.1;	//COM.LC0.CmdGet
      =     #tmpComActive;
//--- New Job
      AN    #CmdNewJob;
      JC    nJob;
      L     0;
      T     #OutTotalWater;	//--> Total weight
//---LC State target commands
nJob: A     #StStarted;	//Set dosing release...
      XN    #Par.OutStateTarget.SetDosingRelease;	// ..if both signals are different
      AN    #CmdFaultReset;
      AN    #CmdNewJob;
      O     #tmpComActive;
      O     #OutRequestActive;
      O     #OutComFault;
      JC    nVal;
      A     #CmdFaultReset;
      =     #Par.OutStateTarget.AlarmReset;
      =     #Par.OutStateTarget.ClearPowerFlag;
      A     #StStarted;
      =     #Par.OutStateTarget.SetDosingRelease;
      A     #CmdNewJob;
      =     #Par.OutStateTarget.ClearErasableTotal;
      JU    CmdS;
//--- New Value
nVal: AN    #CmdNewValue;
      JC    nReq;
      A     #tmpComActive;
      O     #OutComFault;
      O     #OutRequestActive;
      O     #StFault;
      O     #StFalse;
      JC    nReq;
      AN    #Par.OutComFlags.Q_Done;
      AN    #Par.ParComFlags.Without_Q;
      JC    CmdQ;
      AN    #Par.OutComFlags.N_Done;
      AN    #Par.ParComFlags.Without_N;
      JC    CmdN;
      AN    #Par.OutComFlags.X_Done;
      AN    #Par.ParComFlags.Without_X;
      JC    CmdX;
      AN    #Par.OutComFlags.d_Done;
      AN    #Par.ParComFlags.Without_D;
      JC    CmdD;
      AN    #Par.OutComFlags.G_Done;
      AN    #Par.ParComFlags.Without_G;
      JC    CmdG;
      R     #CmdNewValue;
      S     #tmpClearCmdFlag;
//---New Request
nReq: A     #tmpComActive;
      JC    STAT;
      AN    #Par.OutComFlags.d_Done;
      S     #OutRequestActive;
      JC    Cmdd;
      S     #tmpClearCmdFlag;
      R     #OutRequestActive;
      JU    OUT;
NETWORK
TITLE = States
//===State machine===
STAT: A     #StStopped;
      JC    S0;
      A     #StStarted;
      JC    S2;
      A     #StFault;
      JC    S4;
      A     #StFalse;
      JC    S5;
      S     #StStopped;	//Init
      JU    S0;
NETWORK
TITLE =  StStopped
xS0:  S     #StStopped;
      R     #StStarted;
      A     #StFalse;
      O     #StFault;
      R     #StFalse;
      R     #StFault;
      R     #CmdFaultReset;
      R     #OutFaultResetDone;
      L     B#(3, 13);	//Message Operator ('fault cancelled' )
      JC    LOG;
      AN    #tmpReport;
      JC    OUT;
      L     B#(4, 16);	//Message Information ('stopped')
      JU    LOG;
S0:   A     #tmpFault;	//Condition for StFault/StFalse
      JC    xS45;	//StXxx -> StFault transition flag
      A     #tmpOn;
      JC    xS2;
      JU    OUT;
NETWORK
TITLE =  StStarted
xS2:  S     #StStarted;
      R     #StStopped;
      AN    #tmpReport;
      JC    OUT;
      L     B#(4, 17);	//Message Information ('started')
      JU    LOG;
S2:   A     #tmpFault;	//Condition for StFault/StFalse
      JC    xS45;	//StXxx -> StFault transition flag
      A     #tmpOff;
      JC    xS0;
      JU    OUT;
NETWORK
TITLE =  StFault
S4:   AN    #tmpFault;	//---Condition for StStopped
      A     #CmdFaultReset;
      JC    xS0;
      A     #tmpLocal;	//---Condition for StFalse
      JC    xS45;
      A     #OutFaultResetDone;	//reLOG fault
      JC    xS45;
      JU    OUT;
NETWORK
TITLE =  StFalse
//Automatic fault reset
S5:   AN    #tmpFault;	//---Condition for StStopped
      JC    xS0;
      AN    #tmpLocalFault;	//---Condition for StFault
      JC    xS45;	//StXxx -> StFault transition flag
      A     #OutFaultResetDone;	//---Fault reset
      S     #CmdFaultReset;
      R     #OutFaultResetDone;
      JU    OUT;
NETWORK
TITLE = Communication start
Cmdd: S     #Par.OutComFlags.d_Done;
      L     'd';
      JU    GET;
CmdQ: A     #Par.ParComFlags.Without_Q;
      JC    OUT;
      S     #Par.OutComFlags.Q_Done;
      L     'Q';
      JU    PUT;
CmdN: A     #Par.ParComFlags.Without_N;
      JC    OUT;
      S     #Par.OutComFlags.N_Done;
      L     'N';
      JU    PUT;
CmdX: A     #Par.ParComFlags.Without_X;
      JC    OUT;
      S     #Par.OutComFlags.X_Done;
      L     'X';
      JU    PUT;
CmdD: A     #Par.ParComFlags.Without_D;
      JC    OUT;
      S     #Par.OutComFlags.d_Done;
      L     'D';
      JU    PUT;
CmdG: A     #Par.ParComFlags.Without_G;
      JC    OUT;
      S     #Par.OutComFlags.G_Done;
      L     'G';
      JU    PUT;
CmdS: L     'S';
      JU    PUT;
PUT:  SET;
      S     DBX 50.0;	//COM.LC0.CmdPut ;
      JU    ALL1;
GET:  SET;
      S     DBX 50.1;	//COM.LC0.CmdGet ;
ALL1: S     #tmpComActive;
      T     DBB 51;	//COM.LC0.Command;
      JU    OUT;
NETWORK
TITLE = LOG
xS45: S     #tmpClearCmdFlag;	//to clear x_done flags
      R     #StStopped;
      R     #StStarted;
      R     #OutFaultResetDone;
      R     #OutRequestActive;
      A     #InLocal;	//---InLocal=1 -> StFalse -> no LOG message
      S     #StFalse;
      R     #StFault;
      JC    OUT;
      A     #StFault;	// 2.1: Fault flag only when transition -> StFault
      JC    S4J2;
      S     "GCS7_Gr_InFaultFlag";	// 2.1: Gr.InFaultFlag
      CALL  "SYS_Horn_Code" (
           FcCode                   := 1,
           ParObjectType            := 1024,
           ParObjectNo              := #Par.ParObjectNo,
           ParHornCode              := #Par.ParHornCode);
S4J2: SET;	// 2.1:
      S     #StFault;
      R     #StFalse;
      L     B#(1, 14);	//COM communication fault
      A     #OutComFault;
      JC    LOG;
      L     B#(1, 1);
      A     #Par.OutLCAlarm.Ext5NotAvailable;
      JC    LOG;
      L     B#(1, 2);
      A     #Par.OutLCAlarm.Ext24NotAvailable;
      JC    LOG;
      L     B#(1, 3);
      A     #Par.OutLCAlarm.OverloadOutput;
      JC    LOG;
      L     B#(1, 4);
      A     #Par.OutLCAlarm.OverloadOutputOper;
      JC    LOG;
      L     B#(1, 5);
      A     #Par.OutLCAlarm.TurbineFlowFaulty;
      JC    LOG;
      L     B#(1, 6);
      A     #Par.OutLCAlarm.TurbineFlow1Faulty;
      JC    LOG;
      L     B#(1, 7);
      A     #Par.OutLCAlarm.AlarmClosing;
      JC    LOG;
      L     B#(1, 8);
      A     #Par.OutLCAlarm.AlarmOpening;
      JC    LOG;
      L     B#(1, 9);
      A     #Par.OutLCAlarm.NoValidNominalValue;
      JC    LOG;
      L     B#(1, 10);
      A     #Par.OutLCAlarm.ADAlarm;
      JC    LOG;
      L     B#(1, 11);
      A     #Par.OutLCAlarm.InvalidNominalValue;
      JC    LOG;
      L     #OutAlarmNr;
      L     11;
      >I;
      L     B#(1, 15);	//exception error
      JC    LOG;
      L     B#(1, 14);	//COM communication
      JU    LOG;
LOG:  A     #Par.ParLogOff;	//---Set LOG Message
      JC    OUT;
      T     #tmpLOGvalue;
      L     W#16#FF;
      AW;
      T     #OutAlarmNrLog;
      CALL  "GCS7_LogConvert" (
           ObjectNo                 := #Par.ParObjectNo,
           MsgType                  := #Par.ParMsgType,
           ClassMsgTxt              := #tmpLOGvalue,
           OType                    := 1024);	//LOG Message Converter / Entry / Contains Class and TextNo
NETWORK
TITLE = Global End
OUT:  A     #StStarted;
      =     #OutpDosingEnable;
      SET;	//---Clear all commands
      R     #CmdOff;
      R     #CmdOn;
      R     #CmdNext;
      AN    #tmpClearCmdFlag;	//---Clear command flags (x_done)
      JC    STC0;
      R     #Par.OutComFlags.d_Done;
      R     #Par.OutComFlags.Q_Done;
      R     #Par.OutComFlags.N_Done;
      R     #Par.OutComFlags.X_Done;
      R     #Par.OutComFlags.d_Done;
      R     #Par.OutComFlags.G_Done;
//--Output for group 
STC0: AN    #InLocal;
      O     #InManual;
      A     #InDPFault;
      S     "GCS7_Gr_InDPFault";
      AN    #InLocal;
      O     #InManual;
      A     #InHWStop;
      S     "GCS7_Gr_InHWStop";
NETWORK
TITLE = State Code
//--Stopped, Substate ---
      AN    #StStopped;
      JC    STC2;
      L     41;	//Code: StStopped.HWStop
      A     #InHWStop;
      JC    STC;
      L     51;	//Code: StStopped.DPFault
      A     #InDPFault;
      JC    STC;
      L     1;	// Code: stopped
      JC    STC;
//--------------------
STC2: L     3;	//Code: StStarted
      A     #StStarted;
      JC    STC;
      L     5;	//Code: false
      A     #StFalse;
      JC    STC;
      L     32;	//Code: fault
STC:  L     #StCode;	//Old state code
      TAK;
      T     #StCode;	//Save state code
      <>I;
      L     3;	//Load code for CBit methode
      CC    "SYS_CBitCtrl";
NETWORK
TITLE =  Store LC data
      L     #Par.ParLCIdx;
      T     DBW 34;	//COM.Element.Index; 
      L     2;	//Store LC data
      T     DBW 0;	//COM.CODE;
      CDB;
      UC    "GCS7_RS485Ctrl";
      CDB;
END_FUNCTION_BLOCK

